LIN {X 0,Y 298.43,Z 522.305,A -85,B 0,C 180,E1 -16152.517,E2 -16152.517} C_VEL
LIN {X 0,Y 298.415,Z 522.298,A -85,B 0,C 180,E1 -16155.046,E2 -16155.046} C_VEL
LIN {X 0,Y 298.386,Z 522.319,A -85,B 0,C 180,E1 -16158.911,E2 -16158.911} C_VEL
LIN {X 0,Y 298.422,Z 522.312,A -85,B 0,C 180,E1 -16159.614,E2 -16159.614} C_VEL
LIN {X 0,Y 307.334,Z 547.466,A -85,B 0,C 180,E1 -16160.965,E2 -16160.965} C_VEL
LIN {X 0,Y 304.913,Z 622.562,A -85,B 0,C 180,E1 -16163.246,E2 -16163.246} C_VEL
LIN {X 0,Y 304.37,Z 635.953,A -85,B 0,C 180,E1 -16163.915,E2 -16163.915} C_VEL
LIN {X 0,Y 303.565,Z 648.963,A -85,B 0,C 180,E1 -16164.837,E2 -16164.837} C_VEL
LIN {X 0,Y 302.53,Z 662.384,A -85,B 0,C 180,E1 -16166.114,E2 -16166.114} C_VEL
LIN {X 0,Y 301.594,Z 672.65,A -85,B 0,C 180,E1 -16167.354,E2 -16167.354} C_VEL
LIN {X 0,Y 300.607,Z 683.859,A -85,B 0,C 180,E1 -16169.046,E2 -16169.046} C_VEL
LIN {X 0,Y 299.508,Z 693.613,A -85,B 0,C 180,E1 -16170.862,E2 -16170.862} C_VEL
LIN {X 0,Y 298.708,Z 701.527,A -85,B 0,C 180,E1 -16172.69,E2 -16172.69} C_VEL
LIN {X 0,Y 298.005,Z 709.171,A -85,B 0,C 180,E1 -16174.88,E2 -16174.88} C_VEL
LIN {X 0,Y 297.519,Z 715.25,A -85,B 0,C 180,E1 -16177.107,E2 -16177.107} C_VEL
LIN {X 0,Y 297.138,Z 719.644,A -85,B 0,C 180,E1 -16179.219,E2 -16179.219} C_VEL
LIN {X 0,Y 296.954,Z 722.708,A -85,B 0,C 180,E1 -16181.201,E2 -16181.201} C_VEL
LIN {X 0,Y 296.879,Z 725.049,A -85,B 0,C 180,E1 -16183.496,E2 -16183.496} C_VEL
LIN {X 0,Y 297.091,Z 726.196,A -85,B 0,C 180,E1 -16185.9,E2 -16185.9} C_VEL
LIN {X 0,Y 297.35,Z 726.178,A -85,B 0,C 180,E1 -16187.718,E2 -16187.718} C_VEL
LIN {X 0,Y 297.704,Z 725.653,A -85,B 0,C 180,E1 -16189.113,E2 -16189.113} C_VEL
LIN {X 0,Y 298.476,Z 723.763,A -85,B 0,C 180,E1 -16191.463,E2 -16191.463} C_VEL
LIN {X 0,Y 299.56,Z 720.269,A -85,B 0,C 180,E1 -16193.939,E2 -16193.939} C_VEL
LIN {X 0,Y 300.766,Z 716.155,A -85,B 0,C 180,E1 -16195.98,E2 -16195.98} C_VEL
LIN {X 0,Y 302.346,Z 710.28,A -85,B 0,C 180,E1 -16198.196,E2 -16198.196} C_VEL
LIN {X 0,Y 304.151,Z 702.966,A -85,B 0,C 180,E1 -16200.331,E2 -16200.331} C_VEL
LIN {X 0,Y 306.271,Z 694.292,A -85,B 0,C 180,E1 -16202.301,E2 -16202.301} C_VEL
LIN {X 0,Y 308.293,Z 684.485,A -85,B 0,C 180,E1 -16204.085,E2 -16204.085} C_VEL
LIN {X 0,Y 310.321,Z 674.239,A -85,B 0,C 180,E1 -16205.556,E2 -16205.556} C_VEL
LIN {X 0,Y 312.175,Z 663.129,A -85,B 0,C 180,E1 -16206.853,E2 -16206.853} C_VEL
LIN {X 0,Y 313.738,Z 651.807,A -85,B 0,C 180,E1 -16207.886,E2 -16207.886} C_VEL
LIN {X 0,Y 315.086,Z 638.499,A -85,B 0,C 180,E1 -16208.821,E2 -16208.821} C_VEL
LIN {X 0,Y 316.089,Z 625.669,A -85,B 0,C 180,E1 -16209.438,E2 -16209.438} C_VEL
LIN {X 0,Y 318.721,Z 584.023,A -85,B 0,C 180,E1 -16210.836,E2 -16210.836} C_VEL
LIN {X 0,Y 320.456,Z 559.213,A -85,B 0,C 180,E1 -16211.666,E2 -16211.666} C_VEL
LIN {X 0,Y 315.809,Z 550.276,A -85,B 0,C 180,E1 -16212.858,E2 -16212.858} C_VEL
LIN {X 0,Y 310.244,Z 541.034,A -85,B 0,C 180,E1 -16214.366,E2 -16214.366} C_VEL
LIN {X 0,Y 305.459,Z 533.922,A -85,B 0,C 180,E1 -16215.774,E2 -16215.774} C_VEL
LIN {X 0,Y 301.968,Z 529.251,A -85,B 0,C 180,E1 -16216.858,E2 -16216.858} C_VEL
LIN {X 0,Y 299.716,Z 526.202,A -85,B 0,C 180,E1 -16217.617,E2 -16217.617} C_VEL
LIN {X 0,Y 299.533,Z 525.763,A -85,B 0,C 180,E1 -16217.759,E2 -16217.759} C_VEL
LIN {X 0,Y 298.451,Z 522.311,A -85,B 0,C 180,E1 -16220.865,E2 -16220.865} C_VEL
LIN {X 0,Y 298.48,Z 522.303,A -85,B 0,C 180,E1 -16225.076,E2 -16225.076} C_VEL
LIN {X 0,Y 298.464,Z 522.3,A -85,B 0,C 180,E1 -16228.095,E2 -16228.095} C_VEL
LIN {X 0,Y 298.39,Z 522.313,A -85,B 0,C 180,E1 -16232.801,E2 -16232.801} C_VEL
LIN {X 0,Y 298.439,Z 522.308,A -85,B 0,C 180,E1 -16236.808,E2 -16236.808} C_VEL
LIN {X 0,Y 298.384,Z 522.319,A -85,B 0,C 180,E1 -16241.089,E2 -16241.089} C_VEL
LIN {X 0,Y 298.422,Z 522.498,A -85,B 0,C 180,E1 -16243.11,E2 -16243.11} C_VEL
LIN {X 0,Y 299.886,Z 526.896,A -85,B 0,C 180,E1 -16246.594,E2 -16246.594} C_VEL
LIN {X 0,Y 301.229,Z 531.075,A -85,B 0,C 180,E1 -16249.213,E2 -16249.213} C_VEL
LIN {X 0,Y 302.919,Z 536.463,A -85,B 0,C 180,E1 -16252.076,E2 -16252.076} C_VEL
LIN {X 0,Y 304.885,Z 544.324,A -85,B 0,C 180,E1 -16255.578,E2 -16255.578} C_VEL
LIN {X 0,Y 306.272,Z 550.468,A -85,B 0,C 180,E1 -16257.895,E2 -16257.895} C_VEL
LIN {X 0,Y 308.92,Z 555.832,A -85,B 0,C 180,E1 -16258.715,E2 -16258.715} C_VEL
LIN {X 0,Y 311.739,Z 562.313,A -85,B 0,C 180,E1 -16259.566,E2 -16259.566} C_VEL
LIN {X 0,Y 314.455,Z 576.263,A -85,B 0,C 180,E1 -16260.718,E2 -16260.718} C_VEL
LIN {X 0,Y 316.806,Z 593.122,A -85,B 0,C 180,E1 -16261.856,E2 -16261.856} C_VEL
LIN {X 0,Y 317.954,Z 609.201,A -85,B 0,C 180,E1 -16262.737,E2 -16262.737} C_VEL
LIN {X 0,Y 314.374,Z 664.551,A -85,B 0,C 180,E1 -16264.556,E2 -16264.556} C_VEL
LIN {X 0,Y 312.835,Z 678.814,A -85,B 0,C 180,E1 -16265.266,E2 -16265.266} C_VEL
LIN {X 0,Y 310.925,Z 691.732,A -85,B 0,C 180,E1 -16266.17,E2 -16266.17} C_VEL
LIN {X 0,Y 308.588,Z 705.1,A -85,B 0,C 180,E1 -16267.399,E2 -16267.399} C_VEL
LIN {X 0,Y 306.283,Z 716.906,A -85,B 0,C 180,E1 -16268.814,E2 -16268.814} C_VEL
LIN {X 0,Y 304.02,Z 727.605,A -85,B 0,C 180,E1 -16270.416,E2 -16270.416} C_VEL
LIN {X 0,Y 302.162,Z 736.378,A -85,B 0,C 180,E1 -16272.051,E2 -16272.051} C_VEL
LIN {X 0,Y 300.951,Z 742.836,A -85,B 0,C 180,E1 -16273.417,E2 -16273.417} C_VEL
LIN {X 0,Y 299.516,Z 752.316,A -85,B 0,C 180,E1 -16275.39,E2 -16275.39} C_VEL
LIN {X 0,Y 298.286,Z 759.999,A -85,B 0,C 180,E1 -16277.412,E2 -16277.412} C_VEL
LIN {X 0,Y 297.384,Z 767.055,A -85,B 0,C 180,E1 -16279.791,E2 -16279.791} C_VEL
LIN {X 0,Y 296.913,Z 771.726,A -85,B 0,C 180,E1 -16281.835,E2 -16281.835} C_VEL
LIN {X 0,Y 296.63,Z 775.891,A -85,B 0,C 180,E1 -16284.324,E2 -16284.324} C_VEL
LIN {X 0,Y 296.564,Z 777.786,A -85,B 0,C 180,E1 -16285.923,E2 -16285.923} C_VEL
LIN {X 0,Y 296.574,Z 778.942,A -85,B 0,C 180,E1 -16287.284,E2 -16287.284} C_VEL
LIN {X 0,Y 296.524,Z 779.653,A -85,B 0,C 180,E1 -16288.642,E2 -16288.642} C_VEL
LIN {X 0,Y 296.527,Z 779.976,A -85,B 0,C 180,E1 -16290,E2 -16290} C_VEL
LIN {X 0,Y 296.514,Z 779.908,A -85,B 0,C 180,E1 -16291.358,E2 -16291.358} C_VEL
LIN {X 0,Y 296.574,Z 779.416,A -85,B 0,C 180,E1 -16292.716,E2 -16292.716} C_VEL
LIN {X 0,Y 296.565,Z 778.501,A -85,B 0,C 180,E1 -16294.077,E2 -16294.077} C_VEL
LIN {X 0,Y 296.623,Z 776.953,A -85,B 0,C 180,E1 -16295.661,E2 -16295.661} C_VEL
LIN {X 0,Y 296.952,Z 773.26,A -85,B 0,C 180,E1 -16298.164,E2 -16298.164} C_VEL
LIN {X 0,Y 297.447,Z 769.078,A -85,B 0,C 180,E1 -16300.207,E2 -16300.207} C_VEL
LIN {X 0,Y 298.408,Z 762.696,A -85,B 0,C 180,E1 -16302.583,E2 -16302.583} C_VEL
LIN {X 0,Y 299.69,Z 755.711,A -85,B 0,C 180,E1 -16304.601,E2 -16304.601} C_VEL
LIN {X 0,Y 301.202,Z 747.062,A -85,B 0,C 180,E1 -16306.587,E2 -16306.587} C_VEL
LIN {X 0,Y 302.659,Z 737.985,A -85,B 0,C 180,E1 -16308.269,E2 -16308.269} C_VEL
LIN {X 0,Y 304.277,Z 728.064,A -85,B 0,C 180,E1 -16309.742,E2 -16309.742} C_VEL
LIN {X 0,Y 305.903,Z 717.021,A -85,B 0,C 180,E1 -16311.037,E2 -16311.037} C_VEL
LIN {X 0,Y 307.428,Z 704.643,A -85,B 0,C 180,E1 -16312.16,E2 -16312.16} C_VEL
LIN {X 0,Y 308.719,Z 691.932,A -85,B 0,C 180,E1 -16312.989,E2 -16312.989} C_VEL
LIN {X 0,Y 309.686,Z 678.447,A -85,B 0,C 180,E1 -16313.576,E2 -16313.576} C_VEL
LIN {X 0,Y 310.947,Z 632.674,A -85,B 0,C 180,E1 -16314.66,E2 -16314.66} C_VEL
LIN {X 0,Y 311.382,Z 606.3,A -85,B 0,C 180,E1 -16315.281,E2 -16315.281} C_VEL
LIN {X 0,Y 307.249,Z 573.521,A -85,B 0,C 180,E1 -16316.498,E2 -16316.498} C_VEL
LIN {X 0,Y 304.88,Z 559.133,A -85,B 0,C 180,E1 -16317.142,E2 -16317.142} C_VEL
LIN {X 0,Y 304.082,Z 547.632,A -85,B 0,C 180,E1 -16318.209,E2 -16318.209} C_VEL
LIN {X 0,Y 302.745,Z 542.785,A -85,B 0,C 180,E1 -16318.775,E2 -16318.775} C_VEL
LIN {X 0,Y 299.746,Z 528.657,A -85,B 0,C 180,E1 -16322.633,E2 -16322.633} C_VEL
LIN {X 0,Y 298.482,Z 522.306,A -85,B 0,C 180,E1 -16324.454,E2 -16324.454} C_VEL
LIN {X 0,Y 298.405,Z 522.277,A -85,B 0,C 180,E1 -16327.758,E2 -16327.758} C_VEL
LIN {X 0,Y 298.382,Z 522.317,A -85,B 0,C 180,E1 -16331.261,E2 -16331.261} C_VEL
LIN {X 0,Y 298.385,Z 522.314,A -85,B 0,C 180,E1 -16335.041,E2 -16335.041} C_VEL
LIN {X 0,Y 298.415,Z 522.302,A -85,B 0,C 180,E1 -16338.905,E2 -16338.905} C_VEL
LIN {X 0,Y 298.466,Z 522.292,A -85,B 0,C 180,E1 -16343.186,E2 -16343.186} C_VEL
LIN {X 0,Y 298.39,Z 522.312,A -85,B 0,C 180,E1 -16347.199,E2 -16347.199} C_VEL
LIN {X 0,Y 298.426,Z 522.3,A -85,B 0,C 180,E1 -16350.614,E2 -16350.614} C_VEL
LIN {X 0,Y 298.478,Z 522.301,A -85,B 0,C 180,E1 -16353.474,E2 -16353.474} C_VEL
LIN {X 0,Y 298.424,Z 522.288,A -85,B 0,C 180,E1 -16356.699,E2 -16356.699} C_VEL
LIN {X 0,Y 298.531,Z 522.295,A -85,B 0,C 180,E1 -16360.757,E2 -16360.757} C_VEL
LIN {X 0,Y 298.586,Z 522.274,A -85,B 0,C 180,E1 -16364.995,E2 -16364.995} C_VEL
LIN {X 0,Y 298.588,Z 522.283,A -85,B 0,C 180,E1 -16369.147,E2 -16369.147} C_VEL
LIN {X 0,Y 298.749,Z 522.242,A -85,B 0,C 180,E1 -16371.886,E2 -16371.886} C_VEL
LIN {X 0,Y 298.655,Z 522.278,A -85,B 0,C 180,E1 -16374.599,E2 -16374.599} C_VEL
LIN {X 0,Y 298.918,Z 522.229,A -85,B 0,C 180,E1 -16378.653,E2 -16378.653} C_VEL
LIN {X 0,Y 298.918,Z 522.227,A -85,B 0,C 180,E1 -16381.348,E2 -16381.348} C_VEL
LIN {X 0,Y 298.783,Z 522.25,A -85,B 0,C 180,E1 -16386.755,E2 -16386.755} C_VEL
LIN {X 0,Y 298.629,Z 522.264,A -85,B 0,C 180,E1 -16389.482,E2 -16389.482} C_VEL
LIN {X 0,Y 298.546,Z 522.292,A -85,B 0,C 180,E1 -16393.616,E2 -16393.616} C_VEL
LIN {X 0,Y 298.542,Z 522.271,A -85,B 0,C 180,E1 -16396.409,E2 -16396.409} C_VEL
LIN {X 0,Y 298.506,Z 522.302,A -85,B 0,C 180,E1 -16399.655,E2 -16399.655} C_VEL
LIN {X 0,Y 298.452,Z 522.288,A -85,B 0,C 180,E1 -16403.599,E2 -16403.599} C_VEL
LIN {X 0,Y 298.488,Z 522.304,A -85,B 0,C 180,E1 -16406.575,E2 -16406.575} C_VEL
LIN {X 0,Y 298.421,Z 522.296,A -85,B 0,C 180,E1 -16409.641,E2 -16409.641} C_VEL
LIN {X 0,Y 298.394,Z 522.318,A -85,B 0,C 180,E1 -16412.801,E2 -16412.801} C_VEL
LIN {X 0,Y 298.443,Z 522.311,A -85,B 0,C 180,E1 -16416.809,E2 -16416.809} C_VEL
LIN {X 0,Y 298.386,Z 522.32,A -85,B 0,C 180,E1 -16421.089,E2 -16421.089} C_VEL
LIN {X 0,Y 298.387,Z 522.32,A -85,B 0,C 180,E1 -16425.043,E2 -16425.043} C_VEL
LIN {X 0,Y 298.387,Z 522.315,A -85,B 0,C 180,E1 -16428.913,E2 -16428.913} C_VEL
LIN {X 0,Y 298.444,Z 522.313,A -85,B 0,C 180,E1 -16433.194,E2 -16433.194} C_VEL
LIN {X 0,Y 298.469,Z 522.372,A -85,B 0,C 180,E1 -16433.708,E2 -16433.708} C_VEL
LIN {X 0,Y 301.761,Z 534.416,A -85,B 0,C 180,E1 -16436.977,E2 -16436.977} C_VEL
LIN {X 0,Y 304.546,Z 545.909,A -85,B 0,C 180,E1 -16439.874,E2 -16439.874} C_VEL
LIN {X 0,Y 305.469,Z 550.334,A -85,B 0,C 180,E1 -16440.904,E2 -16440.904} C_VEL
LIN {X 0,Y 307.322,Z 555.912,A -85,B 0,C 180,E1 -16441.233,E2 -16441.233} C_VEL
LIN {X 0,Y 312.344,Z 582.163,A -85,B 0,C 180,E1 -16442.382,E2 -16442.382} C_VEL
LIN {X 0,Y 312.661,Z 585.629,A -85,B 0,C 180,E1 -16442.498,E2 -16442.498} C_VEL
LIN {X 0,Y 310.487,Z 661.61,A -85,B 0,C 180,E1 -16444.259,E2 -16444.259} C_VEL
LIN {X 0,Y 309.672,Z 674.686,A -85,B 0,C 180,E1 -16444.817,E2 -16444.817} C_VEL
LIN {X 0,Y 308.672,Z 686.931,A -85,B 0,C 180,E1 -16445.609,E2 -16445.609} C_VEL
LIN {X 0,Y 307.441,Z 698.55,A -85,B 0,C 180,E1 -16446.618,E2 -16446.618} C_VEL
LIN {X 0,Y 305.851,Z 709.944,A -85,B 0,C 180,E1 -16447.898,E2 -16447.898} C_VEL
LIN {X 0,Y 303.969,Z 721.329,A -85,B 0,C 180,E1 -16449.531,E2 -16449.531} C_VEL
LIN {X 0,Y 302.527,Z 729.628,A -85,B 0,C 180,E1 -16451.021,E2 -16451.021} C_VEL
LIN {X 0,Y 301.09,Z 737.273,A -85,B 0,C 180,E1 -16452.687,E2 -16452.687} C_VEL
LIN {X 0,Y 299.86,Z 744.718,A -85,B 0,C 180,E1 -16454.712,E2 -16454.712} C_VEL
LIN {X 0,Y 298.518,Z 751.584,A -85,B 0,C 180,E1 -16457.076,E2 -16457.076} C_VEL
LIN {X 0,Y 297.694,Z 756.111,A -85,B 0,C 180,E1 -16459.114,E2 -16459.114} C_VEL
LIN {X 0,Y 297.33,Z 758.491,A -85,B 0,C 180,E1 -16460.476,E2 -16460.476} C_VEL
LIN {X 0,Y 297.01,Z 760.426,A -85,B 0,C 180,E1 -16461.838,E2 -16461.838} C_VEL
LIN {X 0,Y 296.669,Z 762.838,A -85,B 0,C 180,E1 -16464.256,E2 -16464.256} C_VEL
LIN {X 0,Y 296.596,Z 763.726,A -85,B 0,C 180,E1 -16465.924,E2 -16465.924} C_VEL
LIN {X 0,Y 296.563,Z 764.025,A -85,B 0,C 180,E1 -16467.283,E2 -16467.283} C_VEL
LIN {X 0,Y 296.509,Z 763.946,A -85,B 0,C 180,E1 -16468.642,E2 -16468.642} C_VEL
LIN {X 0,Y 296.524,Z 763.439,A -85,B 0,C 180,E1 -16470,E2 -16470} C_VEL
LIN {X 0,Y 296.753,Z 761.245,A -85,B 0,C 180,E1 -16472.715,E2 -16472.715} C_VEL
LIN {X 0,Y 297.138,Z 758.502,A -85,B 0,C 180,E1 -16474.748,E2 -16474.748} C_VEL
LIN {X 0,Y 297.61,Z 754.749,A -85,B 0,C 180,E1 -16476.781,E2 -16476.781} C_VEL
LIN {X 0,Y 298.284,Z 749.88,A -85,B 0,C 180,E1 -16478.809,E2 -16478.809} C_VEL
LIN {X 0,Y 299.248,Z 743.742,A -85,B 0,C 180,E1 -16480.829,E2 -16480.829} C_VEL
LIN {X 0,Y 300.514,Z 736.035,A -85,B 0,C 180,E1 -16482.836,E2 -16482.836} C_VEL
LIN {X 0,Y 302.039,Z 726.445,A -85,B 0,C 180,E1 -16484.83,E2 -16484.83} C_VEL
LIN {X 0,Y 303.5,Z 716.427,A -85,B 0,C 180,E1 -16486.479,E2 -16486.479} C_VEL
LIN {X 0,Y 304.859,Z 706.554,A -85,B 0,C 180,E1 -16487.785,E2 -16487.785} C_VEL
LIN {X 0,Y 306.131,Z 695.827,A -85,B 0,C 180,E1 -16488.921,E2 -16488.921} C_VEL
LIN {X 0,Y 307.336,Z 684.004,A -85,B 0,C 180,E1 -16489.886,E2 -16489.886} C_VEL
LIN {X 0,Y 308.202,Z 670.49,A -85,B 0,C 180,E1 -16490.679,E2 -16490.679} C_VEL
LIN {X 0,Y 308.801,Z 657.426,A -85,B 0,C 180,E1 -16491.165,E2 -16491.165} C_VEL
LIN {X 0,Y 310.66,Z 582.64,A -85,B 0,C 180,E1 -16492.878,E2 -16492.878} C_VEL
LIN {X 0,Y 305.83,Z 555.571,A -85,B 0,C 180,E1 -16493.97,E2 -16493.97} C_VEL
LIN {X 0,Y 304.741,Z 550.103,A -85,B 0,C 180,E1 -16494.227,E2 -16494.227} C_VEL
LIN {X 0,Y 302.942,Z 540.186,A -85,B 0,C 180,E1 -16496.523,E2 -16496.523} C_VEL
LIN {X 0,Y 300.186,Z 528.619,A -85,B 0,C 180,E1 -16499.449,E2 -16499.449} C_VEL
LIN {X 0,Y 298.436,Z 522.311,A -85,B 0,C 180,E1 -16501.105,E2 -16501.105} C_VEL
LIN {X 0,Y 298.429,Z 522.31,A -85,B 0,C 180,E1 -16504.486,E2 -16504.486} C_VEL
LIN {X 0,Y 298.439,Z 522.31,A -85,B 0,C 180,E1 -16507.753,E2 -16507.753} C_VEL
LIN {X 0,Y 298.451,Z 522.302,A -85,B 0,C 180,E1 -16511.249,E2 -16511.249} C_VEL
LIN {X 0,Y 298.43,Z 522.305,A -85,B 0,C 180,E1 -16512.517,E2 -16512.517} C_VEL
LIN {X 0,Y 297.789,Z 522.392,A -85,B 0,C 180,E1 -16513.644,E2 -16513.644} C_VEL
LIN {X 0,Y 294.902,Z 522.755,A -85,B 0,C 180,E1 -16515.477,E2 -16515.477} C_VEL
LIN {X 0,Y 292.443,Z 523.06,A -85,B 0,C 180,E1 -16516.965,E2 -16516.965} C_VEL
LIN {X 0,Y 291.406,Z 523.188,A -85,B 0,C 180,E1 -16518.12,E2 -16518.12} C_VEL
LIN {X 0,Y 291.332,Z 523.197,A -85,B 0,C 180,E1 -16518.511,E2 -16518.511} C_VEL
LIN {X 0,Y 291.376,Z 523.213,A -85,B 0,C 180,E1 -16519.245,E2 -16519.245} C_VEL
LIN {X 0,Y 300.482,Z 548.952,A -85,B 0,C 180,E1 -16520.636,E2 -16520.636} C_VEL
LIN {X 0,Y 297.989,Z 623.073,A -85,B 0,C 180,E1 -16522.971,E2 -16522.971} C_VEL
LIN {X 0,Y 297.42,Z 636.511,A -85,B 0,C 180,E1 -16523.662,E2 -16523.662} C_VEL
LIN {X 0,Y 296.587,Z 649.592,A -85,B 0,C 180,E1 -16524.614,E2 -16524.614} C_VEL
LIN {X 0,Y 295.526,Z 662.981,A -85,B 0,C 180,E1 -16525.918,E2 -16525.918} C_VEL
LIN {X 0,Y 294.459,Z 674.144,A -85,B 0,C 180,E1 -16527.316,E2 -16527.316} C_VEL
LIN {X 0,Y 293.481,Z 685.006,A -85,B 0,C 180,E1 -16529.012,E2 -16529.012} C_VEL
LIN {X 0,Y 292.394,Z 694.638,A -85,B 0,C 180,E1 -16530.874,E2 -16530.874} C_VEL
LIN {X 0,Y 291.587,Z 702.483,A -85,B 0,C 180,E1 -16532.745,E2 -16532.745} C_VEL
LIN {X 0,Y 290.91,Z 710.082,A -85,B 0,C 180,E1 -16534.989,E2 -16534.989} C_VEL
LIN {X 0,Y 290.409,Z 715.961,A -85,B 0,C 180,E1 -16537.219,E2 -16537.219} C_VEL
LIN {X 0,Y 290.016,Z 720.414,A -85,B 0,C 180,E1 -16539.428,E2 -16539.428} C_VEL
LIN {X 0,Y 289.84,Z 723.632,A -85,B 0,C 180,E1 -16541.625,E2 -16541.625} C_VEL
LIN {X 0,Y 289.785,Z 725.16,A -85,B 0,C 180,E1 -16543.08,E2 -16543.08} C_VEL
LIN {X 0,Y 289.855,Z 726.195,A -85,B 0,C 180,E1 -16544.531,E2 -16544.531} C_VEL
LIN {X 0,Y 290.049,Z 726.754,A -85,B 0,C 180,E1 -16545.977,E2 -16545.977} C_VEL
LIN {X 0,Y 290.242,Z 726.895,A -85,B 0,C 180,E1 -16547.412,E2 -16547.412} C_VEL
LIN {X 0,Y 290.554,Z 726.57,A -85,B 0,C 180,E1 -16548.842,E2 -16548.842} C_VEL
LIN {X 0,Y 291.417,Z 724.833,A -85,B 0,C 180,E1 -16551.401,E2 -16551.401} C_VEL
LIN {X 0,Y 292.445,Z 721.882,A -85,B 0,C 180,E1 -16553.791,E2 -16553.791} C_VEL
LIN {X 0,Y 293.682,Z 718.135,A -85,B 0,C 180,E1 -16555.883,E2 -16555.883} C_VEL
LIN {X 0,Y 295.321,Z 712.655,A -85,B 0,C 180,E1 -16558.16,E2 -16558.16} C_VEL
LIN {X 0,Y 297.181,Z 705.802,A -85,B 0,C 180,E1 -16560.338,E2 -16560.338} C_VEL
LIN {X 0,Y 299.304,Z 697.709,A -85,B 0,C 180,E1 -16562.355,E2 -16562.355} C_VEL
LIN {X 0,Y 301.648,Z 687.639,A -85,B 0,C 180,E1 -16564.342,E2 -16564.342} C_VEL
LIN {X 0,Y 303.8,Z 677.756,A -85,B 0,C 180,E1 -16565.889,E2 -16565.889} C_VEL
LIN {X 0,Y 305.772,Z 666.848,A -85,B 0,C 180,E1 -16567.256,E2 -16567.256} C_VEL
LIN {X 0,Y 307.574,Z 655.47,A -85,B 0,C 180,E1 -16568.376,E2 -16568.376} C_VEL
LIN {X 0,Y 309.044,Z 643.218,A -85,B 0,C 180,E1 -16569.325,E2 -16569.325} C_VEL
LIN {X 0,Y 310.182,Z 630.027,A -85,B 0,C 180,E1 -16570.072,E2 -16570.072} C_VEL
LIN {X 0,Y 311.917,Z 603.449,A -85,B 0,C 180,E1 -16571.032,E2 -16571.032} C_VEL
LIN {X 0,Y 315.065,Z 561.977,A -85,B 0,C 180,E1 -16572.426,E2 -16572.426} C_VEL
LIN {X 0,Y 310.055,Z 552.454,A -85,B 0,C 180,E1 -16573.818,E2 -16573.818} C_VEL
LIN {X 0,Y 304.716,Z 543.622,A -85,B 0,C 180,E1 -16575.389,E2 -16575.389} C_VEL
LIN {X 0,Y 301.575,Z 539.128,A -85,B 0,C 180,E1 -16576.351,E2 -16576.351} C_VEL
LIN {X 0,Y 298.77,Z 535.196,A -85,B 0,C 180,E1 -16577.297,E2 -16577.297} C_VEL
LIN {X 0,Y 295.688,Z 531.254,A -85,B 0,C 180,E1 -16578.358,E2 -16578.358} C_VEL
LIN {X 0,Y 293.052,Z 527.899,A -85,B 0,C 180,E1 -16579.367,E2 -16579.367} C_VEL
LIN {X 0,Y 292.655,Z 527.207,A -85,B 0,C 180,E1 -16579.554,E2 -16579.554} C_VEL
LIN {X 0,Y 291.629,Z 524.342,A -85,B 0,C 180,E1 -16582.68,E2 -16582.68} C_VEL
LIN {X 0,Y 291.394,Z 523.185,A -85,B 0,C 180,E1 -16584.206,E2 -16584.206} C_VEL
LIN {X 0,Y 291.42,Z 523.179,A -85,B 0,C 180,E1 -16587.272,E2 -16587.272} C_VEL
LIN {X 0,Y 291.332,Z 523.189,A -85,B 0,C 180,E1 -16590.437,E2 -16590.437} C_VEL
LIN {X 0,Y 291.339,Z 523.188,A -85,B 0,C 180,E1 -16593.699,E2 -16593.699} C_VEL
LIN {X 0,Y 291.368,Z 523.192,A -85,B 0,C 180,E1 -16597.254,E2 -16597.254} C_VEL
LIN {X 0,Y 291.355,Z 523.201,A -85,B 0,C 180,E1 -16599.679,E2 -16599.679} C_VEL
LIN {X 0,Y 292.076,Z 525.522,A -85,B 0,C 180,E1 -16602.356,E2 -16602.356} C_VEL
LIN {X 0,Y 293.554,Z 529.815,A -85,B 0,C 180,E1 -16606.031,E2 -16606.031} C_VEL
LIN {X 0,Y 295.296,Z 535.352,A -85,B 0,C 180,E1 -16609.605,E2 -16609.605} C_VEL
LIN {X 0,Y 297.112,Z 541.628,A -85,B 0,C 180,E1 -16612.903,E2 -16612.903} C_VEL
LIN {X 0,Y 298.857,Z 548.989,A -85,B 0,C 180,E1 -16616.141,E2 -16616.141} C_VEL
LIN {X 0,Y 301.594,Z 554.384,A -85,B 0,C 180,E1 -16617.094,E2 -16617.094} C_VEL
LIN {X 0,Y 305.364,Z 562.266,A -85,B 0,C 180,E1 -16618.337,E2 -16618.337} C_VEL
LIN {X 0,Y 307.021,Z 566.083,A -85,B 0,C 180,E1 -16618.866,E2 -16618.866} C_VEL
LIN {X 0,Y 309.812,Z 581.74,A -85,B 0,C 180,E1 -16620.17,E2 -16620.17} C_VEL
LIN {X 0,Y 311.638,Z 597.066,A -85,B 0,C 180,E1 -16621.212,E2 -16621.212} C_VEL
LIN {X 0,Y 312.462,Z 610.29,A -85,B 0,C 180,E1 -16621.942,E2 -16621.942} C_VEL
LIN {X 0,Y 308.562,Z 665.089,A -85,B 0,C 180,E1 -16623.814,E2 -16623.814} C_VEL
LIN {X 0,Y 307.037,Z 678.326,A -85,B 0,C 180,E1 -16624.494,E2 -16624.494} C_VEL
LIN {X 0,Y 304.875,Z 692.132,A -85,B 0,C 180,E1 -16625.485,E2 -16625.485} C_VEL
LIN {X 0,Y 302.72,Z 703.718,A -85,B 0,C 180,E1 -16626.574,E2 -16626.574} C_VEL
LIN {X 0,Y 300.52,Z 714.387,A -85,B 0,C 180,E1 -16627.846,E2 -16627.846} C_VEL
LIN {X 0,Y 297.84,Z 726.332,A -85,B 0,C 180,E1 -16629.632,E2 -16629.632} C_VEL
LIN {X 0,Y 295.766,Z 735.251,A -85,B 0,C 180,E1 -16631.29,E2 -16631.29} C_VEL
LIN {X 0,Y 293.634,Z 745.835,A -85,B 0,C 180,E1 -16633.667,E2 -16633.667} C_VEL
LIN {X 0,Y 292.404,Z 753.434,A -85,B 0,C 180,E1 -16635.383,E2 -16635.383} C_VEL
LIN {X 0,Y 291.139,Z 760.858,A -85,B 0,C 180,E1 -16637.452,E2 -16637.452} C_VEL
LIN {X 0,Y 290.383,Z 766.811,A -85,B 0,C 180,E1 -16639.542,E2 -16639.542} C_VEL
LIN {X 0,Y 289.863,Z 771.493,A -85,B 0,C 180,E1 -16641.635,E2 -16641.635} C_VEL
LIN {X 0,Y 289.578,Z 775.046,A -85,B 0,C 180,E1 -16643.73,E2 -16643.73} C_VEL
LIN {X 0,Y 289.466,Z 777.573,A -85,B 0,C 180,E1 -16645.823,E2 -16645.823} C_VEL
LIN {X 0,Y 289.499,Z 778.739,A -85,B 0,C 180,E1 -16647.217,E2 -16647.217} C_VEL
LIN {X 0,Y 289.444,Z 779.456,A -85,B 0,C 180,E1 -16648.609,E2 -16648.609} C_VEL
LIN {X 0,Y 289.444,Z 779.783,A -85,B 0,C 180,E1 -16650,E2 -16650} C_VEL
LIN {X 0,Y 289.435,Z 779.72,A -85,B 0,C 180,E1 -16651.391,E2 -16651.391} C_VEL
LIN {X 0,Y 289.499,Z 779.238,A -85,B 0,C 180,E1 -16652.783,E2 -16652.783} C_VEL
LIN {X 0,Y 289.516,Z 777.021,A -85,B 0,C 180,E1 -16655.572,E2 -16655.572} C_VEL
LIN {X 0,Y 289.742,Z 774.251,A -85,B 0,C 180,E1 -16657.666,E2 -16657.666} C_VEL
LIN {X 0,Y 290.241,Z 770.451,A -85,B 0,C 180,E1 -16659.759,E2 -16659.759} C_VEL
LIN {X 0,Y 290.957,Z 765.509,A -85,B 0,C 180,E1 -16661.848,E2 -16661.848} C_VEL
LIN {X 0,Y 292.089,Z 759.284,A -85,B 0,C 180,E1 -16663.922,E2 -16663.922} C_VEL
LIN {X 0,Y 293.505,Z 751.477,A -85,B 0,C 180,E1 -16665.984,E2 -16665.984} C_VEL
LIN {X 0,Y 295.026,Z 743.072,A -85,B 0,C 180,E1 -16667.769,E2 -16667.769} C_VEL
LIN {X 0,Y 296.593,Z 733.767,A -85,B 0,C 180,E1 -16669.374,E2 -16669.374} C_VEL
LIN {X 0,Y 298.454,Z 722.857,A -85,B 0,C 180,E1 -16670.864,E2 -16670.864} C_VEL
LIN {X 0,Y 299.975,Z 712.158,A -85,B 0,C 180,E1 -16672.015,E2 -16672.015} C_VEL
LIN {X 0,Y 301.401,Z 700.379,A -85,B 0,C 180,E1 -16672.99,E2 -16672.99} C_VEL
LIN {X 0,Y 302.592,Z 687.594,A -85,B 0,C 180,E1 -16673.754,E2 -16673.754} C_VEL
LIN {X 0,Y 303.437,Z 675.041,A -85,B 0,C 180,E1 -16674.229,E2 -16674.229} C_VEL
LIN {X 0,Y 305.091,Z 607.869,A -85,B 0,C 180,E1 -16675.821,E2 -16675.821} C_VEL
LIN {X 0,Y 300.957,Z 574.656,A -85,B 0,C 180,E1 -16677.089,E2 -16677.089} C_VEL
LIN {X 0,Y 298.435,Z 559.219,A -85,B 0,C 180,E1 -16677.782,E2 -16677.782} C_VEL
LIN {X 0,Y 297.976,Z 551.255,A -85,B 0,C 180,E1 -16678.553,E2 -16678.553} C_VEL
LIN {X 0,Y 296.084,Z 544.299,A -85,B 0,C 180,E1 -16679.387,E2 -16679.387} C_VEL
LIN {X 0,Y 294.896,Z 540.06,A -85,B 0,C 180,E1 -16679.936,E2 -16679.936} C_VEL
LIN {X 0,Y 291.912,Z 525.529,A -85,B 0,C 180,E1 -16684.031,E2 -16684.031} C_VEL
LIN {X 0,Y 291.411,Z 523.187,A -85,B 0,C 180,E1 -16684.723,E2 -16684.723} C_VEL
LIN {X 0,Y 291.369,Z 523.156,A -85,B 0,C 180,E1 -16687.252,E2 -16687.252} C_VEL
LIN {X 0,Y 291.33,Z 523.19,A -85,B 0,C 180,E1 -16690.642,E2 -16690.642} C_VEL
LIN {X 0,Y 291.31,Z 523.191,A -85,B 0,C 180,E1 -16694.397,E2 -16694.397} C_VEL
LIN {X 0,Y 291.352,Z 523.18,A -85,B 0,C 180,E1 -16698.397,E2 -16698.397} C_VEL
LIN {X 0,Y 291.376,Z 523.191,A -85,B 0,C 180,E1 -16701.162,E2 -16701.162} C_VEL
LIN {X 0,Y 291.381,Z 523.18,A -85,B 0,C 180,E1 -16704.629,E2 -16704.629} C_VEL
LIN {X 0,Y 291.367,Z 523.182,A -85,B 0,C 180,E1 -16707.95,E2 -16707.95} C_VEL
LIN {X 0,Y 291.377,Z 523.182,A -85,B 0,C 180,E1 -16711.158,E2 -16711.158} C_VEL
LIN {X 0,Y 291.41,Z 523.176,A -85,B 0,C 180,E1 -16714.272,E2 -16714.272} C_VEL
LIN {X 0,Y 291.368,Z 523.172,A -85,B 0,C 180,E1 -16717.299,E2 -16717.299} C_VEL
LIN {X 0,Y 291.452,Z 523.178,A -85,B 0,C 180,E1 -16720.27,E2 -16720.27} C_VEL
LIN {X 0,Y 291.534,Z 523.149,A -85,B 0,C 180,E1 -16724.634,E2 -16724.634} C_VEL
LIN {X 0,Y 291.532,Z 523.165,A -85,B 0,C 180,E1 -16728.881,E2 -16728.881} C_VEL
LIN {X 0,Y 291.7,Z 523.119,A -85,B 0,C 180,E1 -16731.688,E2 -16731.688} C_VEL
LIN {X 0,Y 291.625,Z 523.153,A -85,B 0,C 180,E1 -16734.469,E2 -16734.469} C_VEL
LIN {X 0,Y 291.884,Z 523.105,A -85,B 0,C 180,E1 -16738.621,E2 -16738.621} C_VEL
LIN {X 0,Y 291.885,Z 523.103,A -85,B 0,C 180,E1 -16741.38,E2 -16741.38} C_VEL
LIN {X 0,Y 291.731,Z 523.126,A -85,B 0,C 180,E1 -16746.919,E2 -16746.919} C_VEL
LIN {X 0,Y 291.569,Z 523.146,A -85,B 0,C 180,E1 -16749.714,E2 -16749.714} C_VEL
LIN {X 0,Y 291.516,Z 523.166,A -85,B 0,C 180,E1 -16753.951,E2 -16753.951} C_VEL
LIN {X 0,Y 291.481,Z 523.151,A -85,B 0,C 180,E1 -16756.819,E2 -16756.819} C_VEL
LIN {X 0,Y 291.446,Z 523.18,A -85,B 0,C 180,E1 -16759.876,E2 -16759.876} C_VEL
LIN {X 0,Y 291.395,Z 523.171,A -85,B 0,C 180,E1 -16764.206,E2 -16764.206} C_VEL
LIN {X 0,Y 291.424,Z 523.182,A -85,B 0,C 180,E1 -16767.272,E2 -16767.272} C_VEL
LIN {X 0,Y 291.337,Z 523.182,A -85,B 0,C 180,E1 -16770.437,E2 -16770.437} C_VEL
LIN {X 0,Y 291.342,Z 523.188,A -85,B 0,C 180,E1 -16773.699,E2 -16773.699} C_VEL
LIN {X 0,Y 291.374,Z 523.196,A -85,B 0,C 180,E1 -16777.255,E2 -16777.255} C_VEL
LIN {X 0,Y 291.331,Z 523.194,A -85,B 0,C 180,E1 -16780.643,E2 -16780.643} C_VEL
LIN {X 0,Y 291.312,Z 523.197,A -85,B 0,C 180,E1 -16784.398,E2 -16784.398} C_VEL
LIN {X 0,Y 291.326,Z 523.198,A -85,B 0,C 180,E1 -16788.405,E2 -16788.405} C_VEL
LIN {X 0,Y 291.347,Z 523.194,A -85,B 0,C 180,E1 -16791.159,E2 -16791.159} C_VEL
LIN {X 0,Y 291.398,Z 523.202,A -85,B 0,C 180,E1 -16792.989,E2 -16792.989} C_VEL
LIN {X 0,Y 294.94,Z 535.888,A -85,B 0,C 180,E1 -16796.513,E2 -16796.513} C_VEL
LIN {X 0,Y 298.221,Z 549.592,A -85,B 0,C 180,E1 -16799.993,E2 -16799.993} C_VEL
LIN {X 0,Y 298.422,Z 550.512,A -85,B 0,C 180,E1 -16800.184,E2 -16800.184} C_VEL
LIN {X 0,Y 301.098,Z 557.468,A -85,B 0,C 180,E1 -16800.649,E2 -16800.649} C_VEL
LIN {X 0,Y 306.145,Z 583.989,A -85,B 0,C 180,E1 -16801.846,E2 -16801.846} C_VEL
LIN {X 0,Y 306.194,Z 590.92,A -85,B 0,C 180,E1 -16802.03,E2 -16802.03} C_VEL
LIN {X 0,Y 304.103,Z 660.912,A -85,B 0,C 180,E1 -16803.677,E2 -16803.677} C_VEL
LIN {X 0,Y 303.312,Z 673.642,A -85,B 0,C 180,E1 -16804.204,E2 -16804.204} C_VEL
LIN {X 0,Y 302.348,Z 685.268,A -85,B 0,C 180,E1 -16804.937,E2 -16804.937} C_VEL
LIN {X 0,Y 301.074,Z 697.261,A -85,B 0,C 180,E1 -16805.964,E2 -16805.964} C_VEL
LIN {X 0,Y 299.477,Z 708.638,A -85,B 0,C 180,E1 -16807.219,E2 -16807.219} C_VEL
LIN {X 0,Y 297.922,Z 718.225,A -85,B 0,C 180,E1 -16808.553,E2 -16808.553} C_VEL
LIN {X 0,Y 296.111,Z 727.94,A -85,B 0,C 180,E1 -16810.232,E2 -16810.232} C_VEL
LIN {X 0,Y 294.273,Z 737.353,A -85,B 0,C 180,E1 -16812.273,E2 -16812.273} C_VEL
LIN {X 0,Y 292.949,Z 744.823,A -85,B 0,C 180,E1 -16814.342,E2 -16814.342} C_VEL
LIN {X 0,Y 291.99,Z 749.93,A -85,B 0,C 180,E1 -16816.073,E2 -16816.073} C_VEL
LIN {X 0,Y 290.939,Z 754.854,A -85,B 0,C 180,E1 -16818.152,E2 -16818.152} C_VEL
LIN {X 0,Y 290.298,Z 758.642,A -85,B 0,C 180,E1 -16820.243,E2 -16820.243} C_VEL
LIN {X 0,Y 289.967,Z 760.583,A -85,B 0,C 180,E1 -16821.638,E2 -16821.638} C_VEL
LIN {X 0,Y 289.597,Z 763.127,A -85,B 0,C 180,E1 -16824.273,E2 -16824.273} C_VEL
LIN {X 0,Y 289.497,Z 763.909,A -85,B 0,C 180,E1 -16825.824,E2 -16825.824} C_VEL
LIN {X 0,Y 289.491,Z 764.213,A -85,B 0,C 180,E1 -16827.217,E2 -16827.217} C_VEL
LIN {X 0,Y 289.43,Z 764.14,A -85,B 0,C 180,E1 -16828.609,E2 -16828.609} C_VEL
LIN {X 0,Y 289.441,Z 763.645,A -85,B 0,C 180,E1 -16830,E2 -16830} C_VEL
LIN {X 0,Y 289.681,Z 761.463,A -85,B 0,C 180,E1 -16832.781,E2 -16832.781} C_VEL
LIN {X 0,Y 290.088,Z 758.732,A -85,B 0,C 180,E1 -16834.864,E2 -16834.864} C_VEL
LIN {X 0,Y 290.553,Z 754.993,A -85,B 0,C 180,E1 -16836.946,E2 -16836.946} C_VEL
LIN {X 0,Y 291.274,Z 750.137,A -85,B 0,C 180,E1 -16839.023,E2 -16839.023} C_VEL
LIN {X 0,Y 292.279,Z 744.018,A -85,B 0,C 180,E1 -16841.09,E2 -16841.09} C_VEL
LIN {X 0,Y 293.626,Z 736.332,A -85,B 0,C 180,E1 -16843.143,E2 -16843.143} C_VEL
LIN {X 0,Y 295.207,Z 726.762,A -85,B 0,C 180,E1 -16845.181,E2 -16845.181} C_VEL
LIN {X 0,Y 296.73,Z 716.781,A -85,B 0,C 180,E1 -16846.866,E2 -16846.866} C_VEL
LIN {X 0,Y 298.327,Z 705.568,A -85,B 0,C 180,E1 -16848.366,E2 -16848.366} C_VEL
LIN {X 0,Y 299.615,Z 694.555,A -85,B 0,C 180,E1 -16849.527,E2 -16849.527} C_VEL
LIN {X 0,Y 300.812,Z 683.325,A -85,B 0,C 180,E1 -16850.425,E2 -16850.425} C_VEL
LIN {X 0,Y 301.641,Z 670.512,A -85,B 0,C 180,E1 -16851.184,E2 -16851.184} C_VEL
LIN {X 0,Y 302.266,Z 657.266,A -85,B 0,C 180,E1 -16851.68,E2 -16851.68} C_VEL
LIN {X 0,Y 304.162,Z 583.685,A -85,B 0,C 180,E1 -16853.399,E2 -16853.399} C_VEL
LIN {X 0,Y 299.561,Z 557.431,A -85,B 0,C 180,E1 -16854.485,E2 -16854.485} C_VEL
LIN {X 0,Y 297.973,Z 550.905,A -85,B 0,C 180,E1 -16854.804,E2 -16854.804} C_VEL
LIN {X 0,Y 297.748,Z 550.008,A -85,B 0,C 180,E1 -16854.906,E2 -16854.906} C_VEL
LIN {X 0,Y 295.307,Z 538.033,A -85,B 0,C 180,E1 -16857.786,E2 -16857.786} C_VEL
LIN {X 0,Y 292.412,Z 526.93,A -85,B 0,C 180,E1 -16860.712,E2 -16860.712} C_VEL
LIN {X 0,Y 291.362,Z 523.193,A -85,B 0,C 180,E1 -16861.744,E2 -16861.744} C_VEL
LIN {X 0,Y 291.386,Z 523.189,A -85,B 0,C 180,E1 -16865.37,E2 -16865.37} C_VEL
LIN {X 0,Y 291.378,Z 523.189,A -85,B 0,C 180,E1 -16868.837,E2 -16868.837} C_VEL
LIN {X 0,Y 291.396,Z 523.189,A -85,B 0,C 180,E1 -16872.497,E2 -16872.497} C_VEL
LIN {X 0,Y 291.345,Z 523.184,A -85,B 0,C 180,E1 -16876.357,E2 -16876.357} C_VEL
LIN {X 0,Y 291.332,Z 523.197,A -85,B 0,C 180,E1 -16878.511,E2 -16878.511} C_VEL
LIN {X 0,Y 291.862,Z 523.938,A -85,B 0,C 180,E1 -16878.985,E2 -16878.985} C_VEL
LIN {X 0,Y 293.387,Z 526.274,A -85,B 0,C 180,E1 -16879.44,E2 -16879.44} C_VEL
LIN {X 0,Y 295.583,Z 530.447,A -85,B 0,C 180,E1 -16879.742,E2 -16879.742} C_VEL
LIN {X 0,Y 296.524,Z 534.294,A -85,B 0,C 180,E1 -16879.926,E2 -16879.926} C_VEL
LIN {X 0,Y 296.313,Z 539.044,A -85,B 0,C 180,E1 -16880.045,E2 -16880.045} C_VEL
LIN {X 0,Y 293.571,Z 551.983,A -85,B 0,C 180,E1 -16880.365,E2 -16880.365} C_VEL
LIN {X 0,Y 293.5,Z 553.177,A -85,B 0,C 180,E1 -16880.403,E2 -16880.403} C_VEL
LIN {X 0,Y 291.062,Z 623.382,A -85,B 0,C 180,E1 -16882.677,E2 -16882.677} C_VEL
LIN {X 0,Y 290.431,Z 637.502,A -85,B 0,C 180,E1 -16883.423,E2 -16883.423} C_VEL
LIN {X 0,Y 289.587,Z 650.192,A -85,B 0,C 180,E1 -16884.376,E2 -16884.376} C_VEL
LIN {X 0,Y 288.658,Z 661.851,A -85,B 0,C 180,E1 -16885.523,E2 -16885.523} C_VEL
LIN {X 0,Y 287.668,Z 672.733,A -85,B 0,C 180,E1 -16886.862,E2 -16886.862} C_VEL
LIN {X 0,Y 286.704,Z 682.84,A -85,B 0,C 180,E1 -16888.401,E2 -16888.401} C_VEL
LIN {X 0,Y 285.66,Z 692.156,A -85,B 0,C 180,E1 -16890.135,E2 -16890.135} C_VEL
LIN {X 0,Y 284.786,Z 700.532,A -85,B 0,C 180,E1 -16892.037,E2 -16892.037} C_VEL
LIN {X 0,Y 284.107,Z 707.433,A -85,B 0,C 180,E1 -16893.954,E2 -16893.954} C_VEL
LIN {X 0,Y 283.611,Z 713.053,A -85,B 0,C 180,E1 -16895.866,E2 -16895.866} C_VEL
LIN {X 0,Y 283.119,Z 718.385,A -85,B 0,C 180,E1 -16898.139,E2 -16898.139} C_VEL
LIN {X 0,Y 282.807,Z 722.901,A -85,B 0,C 180,E1 -16900.788,E2 -16900.788} C_VEL
LIN {X 0,Y 282.698,Z 725.139,A -85,B 0,C 180,E1 -16902.643,E2 -16902.643} C_VEL
LIN {X 0,Y 282.74,Z 726.385,A -85,B 0,C 180,E1 -16904.131,E2 -16904.131} C_VEL
LIN {X 0,Y 282.92,Z 727.204,A -85,B 0,C 180,E1 -16905.644,E2 -16905.644} C_VEL
LIN {X 0,Y 283.114,Z 727.502,A -85,B 0,C 180,E1 -16907.09,E2 -16907.09} C_VEL
LIN {X 0,Y 283.427,Z 727.37,A -85,B 0,C 180,E1 -16908.558,E2 -16908.558} C_VEL
LIN {X 0,Y 283.865,Z 726.814,A -85,B 0,C 180,E1 -16910.019,E2 -16910.019} C_VEL
LIN {X 0,Y 284.386,Z 725.794,A -85,B 0,C 180,E1 -16911.473,E2 -16911.473} C_VEL
LIN {X 0,Y 284.973,Z 724.333,A -85,B 0,C 180,E1 -16912.916,E2 -16912.916} C_VEL
LIN {X 0,Y 286.153,Z 721.272,A -85,B 0,C 180,E1 -16915.068,E2 -16915.068} C_VEL
LIN {X 0,Y 287.563,Z 717.109,A -85,B 0,C 180,E1 -16917.198,E2 -16917.198} C_VEL
LIN {X 0,Y 289.215,Z 711.742,A -85,B 0,C 180,E1 -16919.304,E2 -16919.304} C_VEL
LIN {X 0,Y 291.199,Z 705.041,A -85,B 0,C 180,E1 -16921.383,E2 -16921.383} C_VEL
LIN {X 0,Y 293.55,Z 696.588,A -85,B 0,C 180,E1 -16923.431,E2 -16923.431} C_VEL
LIN {X 0,Y 295.649,Z 688.006,A -85,B 0,C 180,E1 -16925.114,E2 -16925.114} C_VEL
LIN {X 0,Y 297.827,Z 678.567,A -85,B 0,C 180,E1 -16926.605,E2 -16926.605} C_VEL
LIN {X 0,Y 299.8,Z 668.467,A -85,B 0,C 180,E1 -16927.918,E2 -16927.918} C_VEL
LIN {X 0,Y 301.955,Z 655.776,A -85,B 0,C 180,E1 -16929.208,E2 -16929.208} C_VEL
LIN {X 0,Y 303.518,Z 643.458,A -85,B 0,C 180,E1 -16930.169,E2 -16930.169} C_VEL
LIN {X 0,Y 304.732,Z 630.126,A -85,B 0,C 180,E1 -16930.926,E2 -16930.926} C_VEL
LIN {X 0,Y 306.971,Z 598.971,A -85,B 0,C 180,E1 -16932.058,E2 -16932.058} C_VEL
LIN {X 0,Y 309.694,Z 564.512,A -85,B 0,C 180,E1 -16933.275,E2 -16933.275} C_VEL
LIN {X 0,Y 304.551,Z 554.913,A -85,B 0,C 180,E1 -16934.794,E2 -16934.794} C_VEL
LIN {X 0,Y 298.902,Z 545.725,A -85,B 0,C 180,E1 -16936.602,E2 -16936.602} C_VEL
LIN {X 0,Y 295.087,Z 540.517,A -85,B 0,C 180,E1 -16937.912,E2 -16937.912} C_VEL
LIN {X 0,Y 292.47,Z 537.054,A -85,B 0,C 180,E1 -16938.892,E2 -16938.892} C_VEL
LIN {X 0,Y 289.223,Z 532.959,A -85,B 0,C 180,E1 -16940.187,E2 -16940.187} C_VEL
LIN {X 0,Y 286.107,Z 529.192,A -85,B 0,C 180,E1 -16941.582,E2 -16941.582} C_VEL
LIN {X 0,Y 285.8,Z 528.644,A -85,B 0,C 180,E1 -16941.835,E2 -16941.835} C_VEL
LIN {X 0,Y 285.135,Z 526.511,A -85,B 0,C 180,E1 -16944.772,E2 -16944.772} C_VEL
LIN {X 0,Y 284.551,Z 525.069,A -85,B 0,C 180,E1 -16947.987,E2 -16947.987} C_VEL
LIN {X 0,Y 284.334,Z 524.39,A -85,B 0,C 180,E1 -16951.269,E2 -16951.269} C_VEL
LIN {X 0,Y 284.437,Z 524.724,A -85,B 0,C 180,E1 -16954.631,E2 -16954.631} C_VEL
LIN {X 0,Y 284.866,Z 526.122,A -85,B 0,C 180,E1 -16958.081,E2 -16958.081} C_VEL
LIN {X 0,Y 285.42,Z 527.515,A -85,B 0,C 180,E1 -16960.244,E2 -16960.244} C_VEL
LIN {X 0,Y 286.402,Z 530.434,A -85,B 0,C 180,E1 -16963.4,E2 -16963.4} C_VEL
LIN {X 0,Y 287.962,Z 534.936,A -85,B 0,C 180,E1 -16967.069,E2 -16967.069} C_VEL
LIN {X 0,Y 289.289,Z 539.488,A -85,B 0,C 180,E1 -16969.93,E2 -16969.93} C_VEL
LIN {X 0,Y 290.865,Z 545.003,A -85,B 0,C 180,E1 -16972.879,E2 -16972.879} C_VEL
LIN {X 0,Y 291.517,Z 547.73,A -85,B 0,C 180,E1 -16974.131,E2 -16974.131} C_VEL
LIN {X 0,Y 294.504,Z 553.323,A -85,B 0,C 180,E1 -16975.311,E2 -16975.311} C_VEL
LIN {X 0,Y 296.056,Z 556.304,A -85,B 0,C 180,E1 -16975.891,E2 -16975.891} C_VEL
LIN {X 0,Y 298.725,Z 561.591,A -85,B 0,C 180,E1 -16976.859,E2 -16976.859} C_VEL
LIN {X 0,Y 301.242,Z 567.049,A -85,B 0,C 180,E1 -16977.722,E2 -16977.722} C_VEL
LIN {X 0,Y 302.404,Z 569.847,A -85,B 0,C 180,E1 -16978.126,E2 -16978.126} C_VEL
LIN {X 0,Y 304.799,Z 584.395,A -85,B 0,C 180,E1 -16979.376,E2 -16979.376} C_VEL
LIN {X 0,Y 306.387,Z 599.003,A -85,B 0,C 180,E1 -16980.403,E2 -16980.403} C_VEL
LIN {X 0,Y 306.993,Z 611.516,A -85,B 0,C 180,E1 -16981.122,E2 -16981.122} C_VEL
LIN {X 0,Y 303.155,Z 663.567,A -85,B 0,C 180,E1 -16982.938,E2 -16982.938} C_VEL
LIN {X 0,Y 301.49,Z 676.862,A -85,B 0,C 180,E1 -16983.618,E2 -16983.618} C_VEL
LIN {X 0,Y 299.536,Z 688.858,A -85,B 0,C 180,E1 -16984.461,E2 -16984.461} C_VEL
LIN {X 0,Y 296.925,Z 702.394,A -85,B 0,C 180,E1 -16985.717,E2 -16985.717} C_VEL
LIN {X 0,Y 294.565,Z 713.228,A -85,B 0,C 180,E1 -16987.003,E2 -16987.003} C_VEL
LIN {X 0,Y 292.223,Z 723.226,A -85,B 0,C 180,E1 -16988.484,E2 -16988.484} C_VEL
LIN {X 0,Y 289.875,Z 732.472,A -85,B 0,C 180,E1 -16990.158,E2 -16990.158} C_VEL
LIN {X 0,Y 287.65,Z 741.592,A -85,B 0,C 180,E1 -16992.203,E2 -16992.203} C_VEL
LIN {X 0,Y 286.514,Z 747.175,A -85,B 0,C 180,E1 -16993.616,E2 -16993.616} C_VEL
LIN {X 0,Y 285.032,Z 755.852,A -85,B 0,C 180,E1 -16995.726,E2 -16995.726} C_VEL
LIN {X 0,Y 283.854,Z 762.743,A -85,B 0,C 180,E1 -16997.851,E2 -16997.851} C_VEL
LIN {X 0,Y 283.138,Z 768.252,A -85,B 0,C 180,E1 -16999.994,E2 -16999.994} C_VEL
LIN {X 0,Y 282.683,Z 772.553,A -85,B 0,C 180,E1 -17002.141,E2 -17002.141} C_VEL
LIN {X 0,Y 282.432,Z 776.001,A -85,B 0,C 180,E1 -17004.475,E2 -17004.475} C_VEL
LIN {X 0,Y 282.402,Z 778.535,A -85,B 0,C 180,E1 -17007.147,E2 -17007.147} C_VEL
LIN {X 0,Y 282.367,Z 779.258,A -85,B 0,C 180,E1 -17008.574,E2 -17008.574} C_VEL
LIN {X 0,Y 282.364,Z 779.59,A -85,B 0,C 180,E1 -17010,E2 -17010} C_VEL
LIN {X 0,Y 282.359,Z 779.531,A -85,B 0,C 180,E1 -17011.426,E2 -17011.426} C_VEL
LIN {X 0,Y 282.402,Z 779.059,A -85,B 0,C 180,E1 -17012.853,E2 -17012.853} C_VEL
LIN {X 0,Y 282.441,Z 776.852,A -85,B 0,C 180,E1 -17015.712,E2 -17015.712} C_VEL
LIN {X 0,Y 282.697,Z 774.093,A -85,B 0,C 180,E1 -17017.859,E2 -17017.859} C_VEL
LIN {X 0,Y 283.206,Z 770.303,A -85,B 0,C 180,E1 -17020.003,E2 -17020.003} C_VEL
LIN {X 0,Y 283.981,Z 765.374,A -85,B 0,C 180,E1 -17022.143,E2 -17022.143} C_VEL
LIN {X 0,Y 285.175,Z 759.163,A -85,B 0,C 180,E1 -17024.267,E2 -17024.267} C_VEL
LIN {X 0,Y 286.668,Z 751.38,A -85,B 0,C 180,E1 -17026.375,E2 -17026.375} C_VEL
LIN {X 0,Y 288.179,Z 743.383,A -85,B 0,C 180,E1 -17028.125,E2 -17028.125} C_VEL
LIN {X 0,Y 289.882,Z 733.715,A -85,B 0,C 180,E1 -17029.841,E2 -17029.841} C_VEL
LIN {X 0,Y 291.829,Z 722.853,A -85,B 0,C 180,E1 -17031.361,E2 -17031.361} C_VEL
LIN {X 0,Y 293.407,Z 712.2,A -85,B 0,C 180,E1 -17032.534,E2 -17032.534} C_VEL
LIN {X 0,Y 294.896,Z 700.488,A -85,B 0,C 180,E1 -17033.527,E2 -17033.527} C_VEL
LIN {X 0,Y 296.129,Z 687.873,A -85,B 0,C 180,E1 -17034.306,E2 -17034.306} C_VEL
LIN {X 0,Y 296.981,Z 675.644,A -85,B 0,C 180,E1 -17034.79,E2 -17034.79} C_VEL
LIN {X 0,Y 298.783,Z 608.778,A -85,B 0,C 180,E1 -17036.405,E2 -17036.405} C_VEL
LIN {X 0,Y 294.696,Z 575.84,A -85,B 0,C 180,E1 -17037.703,E2 -17037.703} C_VEL
LIN {X 0,Y 291.996,Z 559.051,A -85,B 0,C 180,E1 -17038.485,E2 -17038.485} C_VEL
LIN {X 0,Y 291.626,Z 552.823,A -85,B 0,C 180,E1 -17039.12,E2 -17039.12} C_VEL
LIN {X 0,Y 287.112,Z 537.43,A -85,B 0,C 180,E1 -17041.116,E2 -17041.116} C_VEL
LIN {X 0,Y 284.387,Z 524.063,A -85,B 0,C 180,E1 -17045.049,E2 -17045.049} C_VEL
LIN {X 0,Y 284.305,Z 524.031,A -85,B 0,C 180,E1 -17048.169,E2 -17048.169} C_VEL
LIN {X 0,Y 284.267,Z 524.077,A -85,B 0,C 180,E1 -17052.124,E2 -17052.124} C_VEL
LIN {X 0,Y 284.286,Z 524.075,A -85,B 0,C 180,E1 -17056.195,E2 -17056.195} C_VEL
LIN {X 0,Y 284.347,Z 524.065,A -85,B 0,C 180,E1 -17060.012,E2 -17060.012} C_VEL
LIN {X 0,Y 284.35,Z 524.05,A -85,B 0,C 180,E1 -17063.617,E2 -17063.617} C_VEL
LIN {X 0,Y 284.303,Z 524.067,A -85,B 0,C 180,E1 -17067.189,E2 -17067.189} C_VEL
LIN {X 0,Y 284.353,Z 524.051,A -85,B 0,C 180,E1 -17070.376,E2 -17070.376} C_VEL
LIN {X 0,Y 284.372,Z 524.057,A -85,B 0,C 180,E1 -17073.586,E2 -17073.586} C_VEL
LIN {X 0,Y 284.327,Z 524.043,A -85,B 0,C 180,E1 -17076.704,E2 -17076.704} C_VEL
LIN {X 0,Y 284.396,Z 524.049,A -85,B 0,C 180,E1 -17081.261,E2 -17081.261} C_VEL
LIN {X 0,Y 284.472,Z 524.026,A -85,B 0,C 180,E1 -17084.47,E2 -17084.47} C_VEL
LIN {X 0,Y 284.483,Z 524.047,A -85,B 0,C 180,E1 -17088.602,E2 -17088.602} C_VEL
LIN {X 0,Y 284.65,Z 523.997,A -85,B 0,C 180,E1 -17091.481,E2 -17091.481} C_VEL
LIN {X 0,Y 284.595,Z 524.028,A -85,B 0,C 180,E1 -17094.331,E2 -17094.331} C_VEL
LIN {X 0,Y 284.85,Z 523.981,A -85,B 0,C 180,E1 -17098.587,E2 -17098.587} C_VEL
LIN {X 0,Y 284.85,Z 523.979,A -85,B 0,C 180,E1 -17101.414,E2 -17101.414} C_VEL
LIN {X 0,Y 284.681,Z 524.001,A -85,B 0,C 180,E1 -17107.091,E2 -17107.091} C_VEL
LIN {X 0,Y 284.513,Z 524.028,A -85,B 0,C 180,E1 -17109.958,E2 -17109.958} C_VEL
LIN {X 0,Y 284.472,Z 524.04,A -85,B 0,C 180,E1 -17114.304,E2 -17114.304} C_VEL
LIN {X 0,Y 284.419,Z 524.034,A -85,B 0,C 180,E1 -17117.249,E2 -17117.249} C_VEL
LIN {X 0,Y 284.374,Z 524.062,A -85,B 0,C 180,E1 -17120.243,E2 -17120.243} C_VEL
LIN {X 0,Y 284.364,Z 524.043,A -85,B 0,C 180,E1 -17123.876,E2 -17123.876} C_VEL
LIN {X 0,Y 284.362,Z 524.058,A -85,B 0,C 180,E1 -17128.008,E2 -17128.008} C_VEL
LIN {X 0,Y 284.295,Z 524.067,A -85,B 0,C 180,E1 -17131.275,E2 -17131.275} C_VEL
LIN {X 0,Y 284.338,Z 524.056,A -85,B 0,C 180,E1 -17135.349,E2 -17135.349} C_VEL
LIN {X 0,Y 284.31,Z 524.073,A -85,B 0,C 180,E1 -17138.17,E2 -17138.17} C_VEL
LIN {X 0,Y 284.268,Z 524.08,A -85,B 0,C 180,E1 -17142.126,E2 -17142.126} C_VEL
LIN {X 0,Y 284.268,Z 524.074,A -85,B 0,C 180,E1 -17146.193,E2 -17146.193} C_VEL
LIN {X 0,Y 284.306,Z 524.067,A -85,B 0,C 180,E1 -17150.025,E2 -17150.025} C_VEL
LIN {X 0,Y 284.319,Z 524.232,A -85,B 0,C 180,E1 -17152.28,E2 -17152.28} C_VEL
LIN {X 0,Y 287.966,Z 536.8,A -85,B 0,C 180,E1 -17155.853,E2 -17155.853} C_VEL
LIN {X 0,Y 290.645,Z 547.533,A -85,B 0,C 180,E1 -17158.677,E2 -17158.677} C_VEL
LIN {X 0,Y 291.408,Z 550.771,A -85,B 0,C 180,E1 -17159.43,E2 -17159.43} C_VEL
LIN {X 0,Y 295.152,Z 560.167,A -85,B 0,C 180,E1 -17160.099,E2 -17160.099} C_VEL
LIN {X 0,Y 299.984,Z 585.957,A -85,B 0,C 180,E1 -17161.294,E2 -17161.294} C_VEL
LIN {X 0,Y 297.685,Z 661.535,A -85,B 0,C 180,E1 -17163.112,E2 -17163.112} C_VEL
LIN {X 0,Y 296.817,Z 674.83,A -85,B 0,C 180,E1 -17163.692,E2 -17163.692} C_VEL
LIN {X 0,Y 295.711,Z 687.04,A -85,B 0,C 180,E1 -17164.504,E2 -17164.504} C_VEL
LIN {X 0,Y 294.362,Z 699.002,A -85,B 0,C 180,E1 -17165.582,E2 -17165.582} C_VEL
LIN {X 0,Y 292.725,Z 709.918,A -85,B 0,C 180,E1 -17166.85,E2 -17166.85} C_VEL
LIN {X 0,Y 290.915,Z 720.333,A -85,B 0,C 180,E1 -17168.383,E2 -17168.383} C_VEL
LIN {X 0,Y 289.075,Z 729.731,A -85,B 0,C 180,E1 -17170.101,E2 -17170.101} C_VEL
LIN {X 0,Y 287.48,Z 737.429,A -85,B 0,C 180,E1 -17171.839,E2 -17171.839} C_VEL
LIN {X 0,Y 286.12,Z 744.457,A -85,B 0,C 180,E1 -17173.801,E2 -17173.801} C_VEL
LIN {X 0,Y 285.065,Z 750.051,A -85,B 0,C 180,E1 -17175.727,E2 -17175.727} C_VEL
LIN {X 0,Y 283.958,Z 754.991,A -85,B 0,C 180,E1 -17177.856,E2 -17177.856} C_VEL
LIN {X 0,Y 283.282,Z 758.793,A -85,B 0,C 180,E1 -17179.999,E2 -17179.999} C_VEL
LIN {X 0,Y 282.92,Z 760.741,A -85,B 0,C 180,E1 -17181.429,E2 -17181.429} C_VEL
LIN {X 0,Y 282.669,Z 762.28,A -85,B 0,C 180,E1 -17182.859,E2 -17182.859} C_VEL
LIN {X 0,Y 282.485,Z 763.446,A -85,B 0,C 180,E1 -17184.372,E2 -17184.372} C_VEL
LIN {X 0,Y 282.397,Z 764.401,A -85,B 0,C 180,E1 -17187.147,E2 -17187.147} C_VEL
LIN {X 0,Y 282.354,Z 764.334,A -85,B 0,C 180,E1 -17188.574,E2 -17188.574} C_VEL
LIN {X 0,Y 282.361,Z 763.85,A -85,B 0,C 180,E1 -17190,E2 -17190} C_VEL
LIN {X 0,Y 282.612,Z 761.68,A -85,B 0,C 180,E1 -17192.851,E2 -17192.851} C_VEL
LIN {X 0,Y 283.04,Z 758.962,A -85,B 0,C 180,E1 -17194.986,E2 -17194.986} C_VEL
LIN {X 0,Y 283.503,Z 755.237,A -85,B 0,C 180,E1 -17197.12,E2 -17197.12} C_VEL
LIN {X 0,Y 284.268,Z 750.394,A -85,B 0,C 180,E1 -17199.247,E2 -17199.247} C_VEL
LIN {X 0,Y 285.313,Z 744.292,A -85,B 0,C 180,E1 -17201.365,E2 -17201.365} C_VEL
LIN {X 0,Y 286.73,Z 736.629,A -85,B 0,C 180,E1 -17203.465,E2 -17203.465} C_VEL
LIN {X 0,Y 288.389,Z 727.078,A -85,B 0,C 180,E1 -17205.549,E2 -17205.549} C_VEL
LIN {X 0,Y 289.949,Z 717.136,A -85,B 0,C 180,E1 -17207.273,E2 -17207.273} C_VEL
LIN {X 0,Y 291.622,Z 705.954,A -85,B 0,C 180,E1 -17208.804,E2 -17208.804} C_VEL
LIN {X 0,Y 292.956,Z 694.994,A -85,B 0,C 180,E1 -17209.99,E2 -17209.99} C_VEL
LIN {X 0,Y 294.206,Z 683.856,A -85,B 0,C 180,E1 -17210.905,E2 -17210.905} C_VEL
LIN {X 0,Y 295.071,Z 670.981,A -85,B 0,C 180,E1 -17211.689,E2 -17211.689} C_VEL
LIN {X 0,Y 295.731,Z 657.456,A -85,B 0,C 180,E1 -17212.209,E2 -17212.209} C_VEL
LIN {X 0,Y 297.699,Z 584.84,A -85,B 0,C 180,E1 -17213.938,E2 -17213.938} C_VEL
LIN {X 0,Y 293.68,Z 561.219,A -85,B 0,C 180,E1 -17214.936,E2 -17214.936} C_VEL
LIN {X 0,Y 291.969,Z 553.685,A -85,B 0,C 180,E1 -17215.304,E2 -17215.304} C_VEL
LIN {X 0,Y 290.761,Z 550.402,A -85,B 0,C 180,E1 -17215.528,E2 -17215.528} C_VEL
LIN {X 0,Y 288.482,Z 539.574,A -85,B 0,C 180,E1 -17218.186,E2 -17218.186} C_VEL
LIN {X 0,Y 285.635,Z 528.67,A -85,B 0,C 180,E1 -17221.11,E2 -17221.11} C_VEL
LIN {X 0,Y 284.316,Z 524.075,A -85,B 0,C 180,E1 -17222.417,E2 -17222.417} C_VEL
LIN {X 0,Y 284.352,Z 524.058,A -85,B 0,C 180,E1 -17226.382,E2 -17226.382} C_VEL
LIN {X 0,Y 284.351,Z 524.055,A -85,B 0,C 180,E1 -17229.986,E2 -17229.986} C_VEL
LIN {X 0,Y 284.317,Z 524.064,A -85,B 0,C 180,E1 -17233.797,E2 -17233.797} C_VEL
LIN {X 0,Y 284.302,Z 524.071,A -85,B 0,C 180,E1 -17238.129,E2 -17238.129} C_VEL
LIN {X 0,Y 284.31,Z 524.097,A -85,B 0,C 180,E1 -17238.846,E2 -17238.846} C_VEL
LIN {X 0,Y 293.578,Z 550.817,A -85,B 0,C 180,E1 -17240.326,E2 -17240.326} C_VEL
LIN {X 0,Y 293.5,Z 553.177,A -85,B 0,C 180,E1 -17240.403,E2 -17240.403} C_VEL
LIN {X 0,Y 292.694,Z 558.97,A -85,B 0,C 180,E1 -17240.557,E2 -17240.557} C_VEL
LIN {X 0,Y 286.454,Z 577.743,A -85,B 0,C 180,E1 -17240.866,E2 -17240.866} C_VEL
LIN {X 0,Y 285.48,Z 583.539,A -85,B 0,C 180,E1 -17241.017,E2 -17241.017} C_VEL
LIN {X 0,Y 284.106,Z 624.847,A -85,B 0,C 180,E1 -17242.422,E2 -17242.422} C_VEL
LIN {X 0,Y 283.461,Z 638.684,A -85,B 0,C 180,E1 -17243.187,E2 -17243.187} C_VEL
LIN {X 0,Y 282.531,Z 651.835,A -85,B 0,C 180,E1 -17244.227,E2 -17244.227} C_VEL
LIN {X 0,Y 281.484,Z 664.798,A -85,B 0,C 180,E1 -17245.581,E2 -17245.581} C_VEL
LIN {X 0,Y 280.303,Z 676.584,A -85,B 0,C 180,E1 -17247.166,E2 -17247.166} C_VEL
LIN {X 0,Y 279.338,Z 686.435,A -85,B 0,C 180,E1 -17248.804,E2 -17248.804} C_VEL
LIN {X 0,Y 278.355,Z 694.883,A -85,B 0,C 180,E1 -17250.505,E2 -17250.505} C_VEL
LIN {X 0,Y 277.506,Z 702.715,A -85,B 0,C 180,E1 -17252.421,E2 -17252.421} C_VEL
LIN {X 0,Y 276.764,Z 710.618,A -85,B 0,C 180,E1 -17254.827,E2 -17254.827} C_VEL
LIN {X 0,Y 276.261,Z 716.028,A -85,B 0,C 180,E1 -17256.897,E2 -17256.897} C_VEL
LIN {X 0,Y 275.871,Z 720.577,A -85,B 0,C 180,E1 -17259.104,E2 -17259.104} C_VEL
LIN {X 0,Y 275.735,Z 723.059,A -85,B 0,C 180,E1 -17260.649,E2 -17260.649} C_VEL
LIN {X 0,Y 275.647,Z 725.022,A -85,B 0,C 180,E1 -17262.184,E2 -17262.184} C_VEL
LIN {X 0,Y 275.637,Z 726.516,A -85,B 0,C 180,E1 -17263.711,E2 -17263.711} C_VEL
LIN {X 0,Y 275.816,Z 727.622,A -85,B 0,C 180,E1 -17265.522,E2 -17265.522} C_VEL
LIN {X 0,Y 276.294,Z 728.13,A -85,B 0,C 180,E1 -17268.258,E2 -17268.258} C_VEL
LIN {X 0,Y 276.708,Z 727.748,A -85,B 0,C 180,E1 -17269.759,E2 -17269.759} C_VEL
LIN {X 0,Y 277.281,Z 726.907,A -85,B 0,C 180,E1 -17271.293,E2 -17271.293} C_VEL
LIN {X 0,Y 277.853,Z 725.715,A -85,B 0,C 180,E1 -17272.734,E2 -17272.734} C_VEL
LIN {X 0,Y 279.01,Z 722.984,A -85,B 0,C 180,E1 -17274.942,E2 -17274.942} C_VEL
LIN {X 0,Y 280.482,Z 719.179,A -85,B 0,C 180,E1 -17277.127,E2 -17277.127} C_VEL
LIN {X 0,Y 282.211,Z 714.226,A -85,B 0,C 180,E1 -17279.286,E2 -17279.286} C_VEL
LIN {X 0,Y 284.196,Z 707.952,A -85,B 0,C 180,E1 -17281.417,E2 -17281.417} C_VEL
LIN {X 0,Y 286.628,Z 700.058,A -85,B 0,C 180,E1 -17283.514,E2 -17283.514} C_VEL
LIN {X 0,Y 288.84,Z 692.085,A -85,B 0,C 180,E1 -17285.235,E2 -17285.235} C_VEL
LIN {X 0,Y 290.758,Z 684.272,A -85,B 0,C 180,E1 -17286.639,E2 -17286.639} C_VEL
LIN {X 0,Y 293.057,Z 674.291,A -85,B 0,C 180,E1 -17288.099,E2 -17288.099} C_VEL
LIN {X 0,Y 295.294,Z 662.91,A -85,B 0,C 180,E1 -17289.417,E2 -17289.417} C_VEL
LIN {X 0,Y 297.223,Z 650.438,A -85,B 0,C 180,E1 -17290.559,E2 -17290.559} C_VEL
LIN {X 0,Y 298.839,Z 636.757,A -85,B 0,C 180,E1 -17291.488,E2 -17291.488} C_VEL
LIN {X 0,Y 299.981,Z 623.76,A -85,B 0,C 180,E1 -17292.086,E2 -17292.086} C_VEL
LIN {X 0,Y 304.561,Z 567.6,A -85,B 0,C 180,E1 -17294.095,E2 -17294.095} C_VEL
LIN {X 0,Y 299.172,Z 557.477,A -85,B 0,C 180,E1 -17295.829,E2 -17295.829} C_VEL
LIN {X 0,Y 294.605,Z 550.235,A -85,B 0,C 180,E1 -17297.407,E2 -17297.407} C_VEL
LIN {X 0,Y 291.569,Z 545.914,A -85,B 0,C 180,E1 -17298.524,E2 -17298.524} C_VEL
LIN {X 0,Y 289.066,Z 542.592,A -85,B 0,C 180,E1 -17299.518,E2 -17299.518} C_VEL
LIN {X 0,Y 286.446,Z 539.117,A -85,B 0,C 180,E1 -17300.638,E2 -17300.638} C_VEL
LIN {X 0,Y 282.926,Z 534.87,A -85,B 0,C 180,E1 -17302.289,E2 -17302.289} C_VEL
LIN {X 0,Y 279.988,Z 531.774,A -85,B 0,C 180,E1 -17303.854,E2 -17303.854} C_VEL
LIN {X 0,Y 279.207,Z 530.439,A -85,B 0,C 180,E1 -17304.392,E2 -17304.392} C_VEL
LIN {X 0,Y 278.466,Z 528.641,A -85,B 0,C 180,E1 -17308.654,E2 -17308.654} C_VEL
LIN {X 0,Y 278.372,Z 528.255,A -85,B 0,C 180,E1 -17312.018,E2 -17312.018} C_VEL
LIN {X 0,Y 278.545,Z 528.828,A -85,B 0,C 180,E1 -17315.473,E2 -17315.473} C_VEL
LIN {X 0,Y 279.174,Z 530.524,A -85,B 0,C 180,E1 -17319.002,E2 -17319.002} C_VEL
LIN {X 0,Y 280.126,Z 533.421,A -85,B 0,C 180,E1 -17322.64,E2 -17322.64} C_VEL
LIN {X 0,Y 281.586,Z 537.698,A -85,B 0,C 180,E1 -17326.369,E2 -17326.369} C_VEL
LIN {X 0,Y 283.079,Z 542.827,A -85,B 0,C 180,E1 -17329.798,E2 -17329.798} C_VEL
LIN {X 0,Y 284.171,Z 546.332,A -85,B 0,C 180,E1 -17331.687,E2 -17331.687} C_VEL
LIN {X 0,Y 287.594,Z 552.432,A -85,B 0,C 180,E1 -17333.29,E2 -17333.29} C_VEL
LIN {X 0,Y 289.095,Z 555.286,A -85,B 0,C 180,E1 -17333.943,E2 -17333.943} C_VEL
LIN {X 0,Y 292.104,Z 560.896,A -85,B 0,C 180,E1 -17335.168,E2 -17335.168} C_VEL
LIN {X 0,Y 295.177,Z 567.349,A -85,B 0,C 180,E1 -17336.357,E2 -17336.357} C_VEL
LIN {X 0,Y 297.794,Z 573.42,A -85,B 0,C 180,E1 -17337.329,E2 -17337.329} C_VEL
LIN {X 0,Y 299.865,Z 586.874,A -85,B 0,C 180,E1 -17338.53,E2 -17338.53} C_VEL
LIN {X 0,Y 301.253,Z 601.096,A -85,B 0,C 180,E1 -17339.562,E2 -17339.562} C_VEL
LIN {X 0,Y 301.741,Z 612.617,A -85,B 0,C 180,E1 -17340.238,E2 -17340.238} C_VEL
LIN {X 0,Y 297.693,Z 663.1,A -85,B 0,C 180,E1 -17342.065,E2 -17342.065} C_VEL
LIN {X 0,Y 295.843,Z 676.95,A -85,B 0,C 180,E1 -17342.788,E2 -17342.788} C_VEL
LIN {X 0,Y 293.639,Z 689.659,A -85,B 0,C 180,E1 -17343.719,E2 -17343.719} C_VEL
LIN {X 0,Y 290.897,Z 702.836,A -85,B 0,C 180,E1 -17344.989,E2 -17344.989} C_VEL
LIN {X 0,Y 288.139,Z 714.499,A -85,B 0,C 180,E1 -17346.46,E2 -17346.46} C_VEL
LIN {X 0,Y 285.194,Z 726.109,A -85,B 0,C 180,E1 -17348.307,E2 -17348.307} C_VEL
LIN {X 0,Y 282.86,Z 734.768,A -85,B 0,C 180,E1 -17350.024,E2 -17350.024} C_VEL
LIN {X 0,Y 280.543,Z 743.481,A -85,B 0,C 180,E1 -17352.167,E2 -17352.167} C_VEL
LIN {X 0,Y 279.381,Z 748.505,A -85,B 0,C 180,E1 -17353.561,E2 -17353.561} C_VEL
LIN {X 0,Y 277.883,Z 756.821,A -85,B 0,C 180,E1 -17355.725,E2 -17355.725} C_VEL
LIN {X 0,Y 276.721,Z 763.5,A -85,B 0,C 180,E1 -17357.906,E2 -17357.906} C_VEL
LIN {X 0,Y 275.921,Z 769.597,A -85,B 0,C 180,E1 -17360.47,E2 -17360.47} C_VEL
LIN {X 0,Y 275.515,Z 773.532,A -85,B 0,C 180,E1 -17362.673,E2 -17362.673} C_VEL
LIN {X 0,Y 275.354,Z 776.003,A -85,B 0,C 180,E1 -17364.513,E2 -17364.513} C_VEL
LIN {X 0,Y 275.308,Z 778.33,A -85,B 0,C 180,E1 -17367.074,E2 -17367.074} C_VEL
LIN {X 0,Y 275.291,Z 779.06,A -85,B 0,C 180,E1 -17368.537,E2 -17368.537} C_VEL
LIN {X 0,Y 275.285,Z 779.397,A -85,B 0,C 180,E1 -17370,E2 -17370} C_VEL
LIN {X 0,Y 275.284,Z 779.343,A -85,B 0,C 180,E1 -17371.463,E2 -17371.463} C_VEL
LIN {X 0,Y 275.308,Z 778.88,A -85,B 0,C 180,E1 -17372.926,E2 -17372.926} C_VEL
LIN {X 0,Y 275.349,Z 776.683,A -85,B 0,C 180,E1 -17375.86,E2 -17375.86} C_VEL
LIN {X 0,Y 275.65,Z 773.934,A -85,B 0,C 180,E1 -17378.061,E2 -17378.061} C_VEL
LIN {X 0,Y 276.189,Z 770.156,A -85,B 0,C 180,E1 -17380.26,E2 -17380.26} C_VEL
LIN {X 0,Y 276.994,Z 765.239,A -85,B 0,C 180,E1 -17382.454,E2 -17382.454} C_VEL
LIN {X 0,Y 278.279,Z 759.043,A -85,B 0,C 180,E1 -17384.628,E2 -17384.628} C_VEL
LIN {X 0,Y 279.855,Z 751.284,A -85,B 0,C 180,E1 -17386.786,E2 -17386.786} C_VEL
LIN {X 0,Y 281.541,Z 742.636,A -85,B 0,C 180,E1 -17388.711,E2 -17388.711} C_VEL
LIN {X 0,Y 283.433,Z 732.602,A -85,B 0,C 180,E1 -17390.502,E2 -17390.502} C_VEL
LIN {X 0,Y 285.454,Z 721.44,A -85,B 0,C 180,E1 -17392.052,E2 -17392.052} C_VEL
LIN {X 0,Y 287.108,Z 710.503,A -85,B 0,C 180,E1 -17393.248,E2 -17393.248} C_VEL
LIN {X 0,Y 288.702,Z 698.362,A -85,B 0,C 180,E1 -17394.254,E2 -17394.254} C_VEL
LIN {X 0,Y 289.916,Z 685.526,A -85,B 0,C 180,E1 -17395.005,E2 -17395.005} C_VEL
LIN {X 0,Y 290.715,Z 671.974,A -85,B 0,C 180,E1 -17395.506,E2 -17395.506} C_VEL
LIN {X 0,Y 292.451,Z 609.507,A -85,B 0,C 180,E1 -17397.025,E2 -17397.025} C_VEL
LIN {X 0,Y 288.478,Z 576.908,A -85,B 0,C 180,E1 -17398.346,E2 -17398.346} C_VEL
LIN {X 0,Y 285.563,Z 558.93,A -85,B 0,C 180,E1 -17399.212,E2 -17399.212} C_VEL
LIN {X 0,Y 285.217,Z 554.458,A -85,B 0,C 180,E1 -17399.705,E2 -17399.705} C_VEL
LIN {X 0,Y 280.32,Z 538.261,A -85,B 0,C 180,E1 -17401.916,E2 -17401.916} C_VEL
LIN {X 0,Y 279.236,Z 534.346,A -85,B 0,C 180,E1 -17402.491,E2 -17402.491} C_VEL
LIN {X 0,Y 277.333,Z 524.938,A -85,B 0,C 180,E1 -17405.372,E2 -17405.372} C_VEL
LIN {X 0,Y 277.23,Z 524.919,A -85,B 0,C 180,E1 -17409.328,E2 -17409.328} C_VEL
LIN {X 0,Y 277.213,Z 524.946,A -85,B 0,C 180,E1 -17413.196,E2 -17413.196} C_VEL
LIN {X 0,Y 277.237,Z 524.943,A -85,B 0,C 180,E1 -17417.319,E2 -17417.319} C_VEL
LIN {X 0,Y 277.263,Z 524.949,A -85,B 0,C 180,E1 -17420.677,E2 -17420.677} C_VEL
LIN {X 0,Y 277.301,Z 524.931,A -85,B 0,C 180,E1 -17424.344,E2 -17424.344} C_VEL
LIN {X 0,Y 277.239,Z 524.942,A -85,B 0,C 180,E1 -17427.836,E2 -17427.836} C_VEL
LIN {X 0,Y 277.284,Z 524.938,A -85,B 0,C 180,E1 -17431.212,E2 -17431.212} C_VEL
LIN {X 0,Y 277.304,Z 524.928,A -85,B 0,C 180,E1 -17434.479,E2 -17434.479} C_VEL
LIN {X 0,Y 277.262,Z 524.933,A -85,B 0,C 180,E1 -17437.653,E2 -17437.653} C_VEL
LIN {X 0,Y 277.338,Z 524.934,A -85,B 0,C 180,E1 -17440.766,E2 -17440.766} C_VEL
LIN {X 0,Y 277.422,Z 524.912,A -85,B 0,C 180,E1 -17445.325,E2 -17445.325} C_VEL
LIN {X 0,Y 277.501,Z 524.905,A -85,B 0,C 180,E1 -17449.789,E2 -17449.789} C_VEL
LIN {X 0,Y 277.644,Z 524.875,A -85,B 0,C 180,E1 -17452.729,E2 -17452.729} C_VEL
LIN {X 0,Y 277.816,Z 524.857,A -85,B 0,C 180,E1 -17458.551,E2 -17458.551} C_VEL
LIN {X 0,Y 277.816,Z 524.854,A -85,B 0,C 180,E1 -17461.45,E2 -17461.45} C_VEL
LIN {X 0,Y 277.636,Z 524.877,A -85,B 0,C 180,E1 -17467.272,E2 -17467.272} C_VEL
LIN {X 0,Y 277.455,Z 524.91,A -85,B 0,C 180,E1 -17470.214,E2 -17470.214} C_VEL
LIN {X 0,Y 277.423,Z 524.911,A -85,B 0,C 180,E1 -17474.675,E2 -17474.675} C_VEL
LIN {X 0,Y 277.34,Z 524.938,A -85,B 0,C 180,E1 -17479.235,E2 -17479.235} C_VEL
LIN {X 0,Y 277.315,Z 524.923,A -85,B 0,C 180,E1 -17484.171,E2 -17484.171} C_VEL
LIN {X 0,Y 277.333,Z 524.935,A -85,B 0,C 180,E1 -17487.51,E2 -17487.51} C_VEL
LIN {X 0,Y 277.269,Z 524.934,A -85,B 0,C 180,E1 -17490.482,E2 -17490.482} C_VEL
LIN {X 0,Y 277.244,Z 524.943,A -85,B 0,C 180,E1 -17493.897,E2 -17493.897} C_VEL
LIN {X 0,Y 277.265,Z 524.952,A -85,B 0,C 180,E1 -17497.47,E2 -17497.47} C_VEL
LIN {X 0,Y 277.208,Z 524.959,A -85,B 0,C 180,E1 -17501.238,E2 -17501.238} C_VEL
LIN {X 0,Y 277.216,Z 524.959,A -85,B 0,C 180,E1 -17505.224,E2 -17505.224} C_VEL
LIN {X 0,Y 277.222,Z 524.949,A -85,B 0,C 180,E1 -17509.513,E2 -17509.513} C_VEL
LIN {X 0,Y 277.264,Z 525.082,A -85,B 0,C 180,E1 -17511.453,E2 -17511.453} C_VEL
LIN {X 0,Y 280.74,Z 536.673,A -85,B 0,C 180,E1 -17514.847,E2 -17514.847} C_VEL
LIN {X 0,Y 283.634,Z 548.159,A -85,B 0,C 180,E1 -17517.964,E2 -17517.964} C_VEL
LIN {X 0,Y 284.354,Z 550.994,A -85,B 0,C 180,E1 -17518.627,E2 -17518.627} C_VEL
LIN {X 0,Y 289.19,Z 562.566,A -85,B 0,C 180,E1 -17519.512,E2 -17519.512} C_VEL
LIN {X 0,Y 293.701,Z 586.865,A -85,B 0,C 180,E1 -17520.673,E2 -17520.673} C_VEL
LIN {X 0,Y 291.285,Z 662.161,A -85,B 0,C 180,E1 -17522.521,E2 -17522.521} C_VEL
LIN {X 0,Y 290.393,Z 675.254,A -85,B 0,C 180,E1 -17523.111,E2 -17523.111} C_VEL
LIN {X 0,Y 289.223,Z 687.734,A -85,B 0,C 180,E1 -17523.966,E2 -17523.966} C_VEL
LIN {X 0,Y 287.844,Z 699.243,A -85,B 0,C 180,E1 -17525.029,E2 -17525.029} C_VEL
LIN {X 0,Y 286.199,Z 709.906,A -85,B 0,C 180,E1 -17526.29,E2 -17526.29} C_VEL
LIN {X 0,Y 284.321,Z 720.357,A -85,B 0,C 180,E1 -17527.855,E2 -17527.855} C_VEL
LIN {X 0,Y 282.385,Z 729.784,A -85,B 0,C 180,E1 -17529.609,E2 -17529.609} C_VEL
LIN {X 0,Y 280.718,Z 737.505,A -85,B 0,C 180,E1 -17531.386,E2 -17531.386} C_VEL
LIN {X 0,Y 279.227,Z 744.768,A -85,B 0,C 180,E1 -17533.46,E2 -17533.46} C_VEL
LIN {X 0,Y 278.159,Z 750.172,A -85,B 0,C 180,E1 -17535.365,E2 -17535.365} C_VEL
LIN {X 0,Y 276.993,Z 755.128,A -85,B 0,C 180,E1 -17537.546,E2 -17537.546} C_VEL
LIN {X 0,Y 276.25,Z 758.944,A -85,B 0,C 180,E1 -17539.742,E2 -17539.742} C_VEL
LIN {X 0,Y 275.892,Z 760.898,A -85,B 0,C 180,E1 -17541.209,E2 -17541.209} C_VEL
LIN {X 0,Y 275.607,Z 762.444,A -85,B 0,C 180,E1 -17542.675,E2 -17542.675} C_VEL
LIN {X 0,Y 275.377,Z 763.752,A -85,B 0,C 180,E1 -17544.47,E2 -17544.47} C_VEL
LIN {X 0,Y 275.306,Z 764.589,A -85,B 0,C 180,E1 -17547.074,E2 -17547.074} C_VEL
LIN {X 0,Y 275.279,Z 764.527,A -85,B 0,C 180,E1 -17548.537,E2 -17548.537} C_VEL
LIN {X 0,Y 275.283,Z 764.056,A -85,B 0,C 180,E1 -17550,E2 -17550} C_VEL
LIN {X 0,Y 275.546,Z 761.898,A -85,B 0,C 180,E1 -17552.924,E2 -17552.924} C_VEL
LIN {X 0,Y 275.973,Z 759.192,A -85,B 0,C 180,E1 -17555.114,E2 -17555.114} C_VEL
LIN {X 0,Y 276.635,Z 754.561,A -85,B 0,C 180,E1 -17557.77,E2 -17557.77} C_VEL
LIN {X 0,Y 277.616,Z 748.759,A -85,B 0,C 180,E1 -17560.207,E2 -17560.207} C_VEL
LIN {X 0,Y 278.801,Z 742.188,A -85,B 0,C 180,E1 -17562.372,E2 -17562.372} C_VEL
LIN {X 0,Y 280.382,Z 734.005,A -85,B 0,C 180,E1 -17564.516,E2 -17564.516} C_VEL
LIN {X 0,Y 281.9,Z 725.568,A -85,B 0,C 180,E1 -17566.288,E2 -17566.288} C_VEL
LIN {X 0,Y 283.389,Z 716.355,A -85,B 0,C 180,E1 -17567.872,E2 -17567.872} C_VEL
LIN {X 0,Y 284.937,Z 706.34,A -85,B 0,C 180,E1 -17569.262,E2 -17569.262} C_VEL
LIN {X 0,Y 286.318,Z 695.426,A -85,B 0,C 180,E1 -17570.474,E2 -17570.474} C_VEL
LIN {X 0,Y 287.617,Z 684.386,A -85,B 0,C 180,E1 -17571.407,E2 -17571.407} C_VEL
LIN {X 0,Y 288.536,Z 671.209,A -85,B 0,C 180,E1 -17572.23,E2 -17572.23} C_VEL
LIN {X 0,Y 289.186,Z 658.654,A -85,B 0,C 180,E1 -17572.732,E2 -17572.732} C_VEL
LIN {X 0,Y 291.284,Z 585.978,A -85,B 0,C 180,E1 -17574.5,E2 -17574.5} C_VEL
LIN {X 0,Y 287.389,Z 562.746,A -85,B 0,C 180,E1 -17575.51,E2 -17575.51} C_VEL
LIN {X 0,Y 285.957,Z 556.353,A -85,B 0,C 180,E1 -17575.83,E2 -17575.83} C_VEL
LIN {X 0,Y 283.694,Z 550.48,A -85,B 0,C 180,E1 -17576.251,E2 -17576.251} C_VEL
LIN {X 0,Y 281.283,Z 539.584,A -85,B 0,C 180,E1 -17579.014,E2 -17579.014} C_VEL
LIN {X 0,Y 278.328,Z 528.695,A -85,B 0,C 180,E1 -17582.023,E2 -17582.023} C_VEL
LIN {X 0,Y 277.253,Z 524.947,A -85,B 0,C 180,E1 -17583.099,E2 -17583.099} C_VEL
LIN {X 0,Y 277.326,Z 524.936,A -85,B 0,C 180,E1 -17585.811,E2 -17585.811} C_VEL
LIN {X 0,Y 277.266,Z 524.942,A -85,B 0,C 180,E1 -17589.322,E2 -17589.322} C_VEL
LIN {X 0,Y 277.262,Z 524.947,A -85,B 0,C 180,E1 -17593.186,E2 -17593.186} C_VEL
LIN {X 0,Y 277.231,Z 524.952,A -85,B 0,C 180,E1 -17597.32,E2 -17597.32} C_VEL
LIN {X 0,Y 277.302,Z 525.057,A -85,B 0,C 180,E1 -17598.44,E2 -17598.44} C_VEL
LIN {X 0,Y 286.596,Z 551.432,A -85,B 0,C 180,E1 -17599.955,E2 -17599.955} C_VEL
LIN {X 0,Y 285.48,Z 583.539,A -85,B 0,C 180,E1 -17601.017,E2 -17601.017} C_VEL
LIN {X 0,Y 284.52,Z 589.327,A -85,B 0,C 180,E1 -17601.168,E2 -17601.168} C_VEL
LIN {X 0,Y 278.392,Z 608.092,A -85,B 0,C 180,E1 -17601.525,E2 -17601.525} C_VEL
LIN {X 0,Y 277.544,Z 613.877,A -85,B 0,C 180,E1 -17601.694,E2 -17601.694} C_VEL
LIN {X 0,Y 276.938,Z 629.409,A -85,B 0,C 180,E1 -17602.332,E2 -17602.332} C_VEL
LIN {X 0,Y 276.174,Z 643.901,A -85,B 0,C 180,E1 -17603.271,E2 -17603.271} C_VEL
LIN {X 0,Y 275.269,Z 655.997,A -85,B 0,C 180,E1 -17604.345,E2 -17604.345} C_VEL
LIN {X 0,Y 274.054,Z 669.236,A -85,B 0,C 180,E1 -17605.876,E2 -17605.876} C_VEL
LIN {X 0,Y 272.894,Z 680.716,A -85,B 0,C 180,E1 -17607.58,E2 -17607.58} C_VEL
LIN {X 0,Y 271.869,Z 690.125,A -85,B 0,C 180,E1 -17609.299,E2 -17609.299} C_VEL
LIN {X 0,Y 270.851,Z 699.499,A -85,B 0,C 180,E1 -17611.396,E2 -17611.396} C_VEL
LIN {X 0,Y 269.972,Z 707.808,A -85,B 0,C 180,E1 -17613.733,E2 -17613.733} C_VEL
LIN {X 0,Y 269.391,Z 714.09,A -85,B 0,C 180,E1 -17615.934,E2 -17615.934} C_VEL
LIN {X 0,Y 268.863,Z 719.863,A -85,B 0,C 180,E1 -17618.533,E2 -17618.533} C_VEL
LIN {X 0,Y 268.665,Z 722.94,A -85,B 0,C 180,E1 -17620.339,E2 -17620.339} C_VEL
LIN {X 0,Y 268.58,Z 724.813,A -85,B 0,C 180,E1 -17621.699,E2 -17621.699} C_VEL
LIN {X 0,Y 268.537,Z 726.48,A -85,B 0,C 180,E1 -17623.268,E2 -17623.268} C_VEL
LIN {X 0,Y 268.729,Z 728.02,A -85,B 0,C 180,E1 -17625.381,E2 -17625.381} C_VEL
LIN {X 0,Y 269.138,Z 728.747,A -85,B 0,C 180,E1 -17627.941,E2 -17627.941} C_VEL
LIN {X 0,Y 269.557,Z 728.599,A -85,B 0,C 180,E1 -17629.484,E2 -17629.484} C_VEL
LIN {X 0,Y 270.192,Z 727.866,A -85,B 0,C 180,E1 -17631.264,E2 -17631.264} C_VEL
LIN {X 0,Y 271.464,Z 725.49,A -85,B 0,C 180,E1 -17634.056,E2 -17634.056} C_VEL
LIN {X 0,Y 272.873,Z 722.406,A -85,B 0,C 180,E1 -17636.308,E2 -17636.308} C_VEL
LIN {X 0,Y 274.549,Z 718.224,A -85,B 0,C 180,E1 -17638.533,E2 -17638.533} C_VEL
LIN {X 0,Y 276.516,Z 712.835,A -85,B 0,C 180,E1 -17640.728,E2 -17640.728} C_VEL
LIN {X 0,Y 278.831,Z 706.073,A -85,B 0,C 180,E1 -17642.889,E2 -17642.889} C_VEL
LIN {X 0,Y 281.533,Z 697.608,A -85,B 0,C 180,E1 -17645.012,E2 -17645.012} C_VEL
LIN {X 0,Y 284.088,Z 688.363,A -85,B 0,C 180,E1 -17646.878,E2 -17646.878} C_VEL
LIN {X 0,Y 286.881,Z 677.224,A -85,B 0,C 180,E1 -17648.63,E2 -17648.63} C_VEL
LIN {X 0,Y 289.233,Z 666.602,A -85,B 0,C 180,E1 -17649.97,E2 -17649.97} C_VEL
LIN {X 0,Y 291.291,Z 655.014,A -85,B 0,C 180,E1 -17651.129,E2 -17651.129} C_VEL
LIN {X 0,Y 293.225,Z 640.933,A -85,B 0,C 180,E1 -17652.193,E2 -17652.193} C_VEL
LIN {X 0,Y 294.531,Z 627.59,A -85,B 0,C 180,E1 -17652.883,E2 -17652.883} C_VEL
LIN {X 0,Y 298.87,Z 577.908,A -85,B 0,C 180,E1 -17654.721,E2 -17654.721} C_VEL
LIN {X 0,Y 299.492,Z 570.448,A -85,B 0,C 180,E1 -17655.013,E2 -17655.013} C_VEL
LIN {X 0,Y 295.007,Z 562.028,A -85,B 0,C 180,E1 -17656.549,E2 -17656.549} C_VEL
LIN {X 0,Y 291.06,Z 555.64,A -85,B 0,C 180,E1 -17657.988,E2 -17657.988} C_VEL
LIN {X 0,Y 286.923,Z 549.528,A -85,B 0,C 180,E1 -17659.664,E2 -17659.664} C_VEL
LIN {X 0,Y 283.722,Z 545.325,A -85,B 0,C 180,E1 -17661.087,E2 -17661.087} C_VEL
LIN {X 0,Y 280.431,Z 541.237,A -85,B 0,C 180,E1 -17662.715,E2 -17662.715} C_VEL
LIN {X 0,Y 277.375,Z 537.766,A -85,B 0,C 180,E1 -17664.443,E2 -17664.443} C_VEL
LIN {X 0,Y 276.728,Z 536.918,A -85,B 0,C 180,E1 -17664.866,E2 -17664.866} C_VEL
LIN {X 0,Y 273.438,Z 533.937,A -85,B 0,C 180,E1 -17667.143,E2 -17667.143} C_VEL
LIN {X 0,Y 272.562,Z 532.608,A -85,B 0,C 180,E1 -17668.07,E2 -17668.07} C_VEL
LIN {X 0,Y 272.403,Z 532.088,A -85,B 0,C 180,E1 -17671.638,E2 -17671.638} C_VEL
LIN {X 0,Y 272.49,Z 532.482,A -85,B 0,C 180,E1 -17674.57,E2 -17674.57} C_VEL
LIN {X 0,Y 272.973,Z 533.883,A -85,B 0,C 180,E1 -17678.163,E2 -17678.163} C_VEL
LIN {X 0,Y 273.899,Z 536.6,A -85,B 0,C 180,E1 -17681.918,E2 -17681.918} C_VEL
LIN {X 0,Y 275.229,Z 540.477,A -85,B 0,C 180,E1 -17685.642,E2 -17685.642} C_VEL
LIN {X 0,Y 276.362,Z 544.194,A -85,B 0,C 180,E1 -17688.285,E2 -17688.285} C_VEL
LIN {X 0,Y 280.24,Z 550.851,A -85,B 0,C 180,E1 -17690.624,E2 -17690.624} C_VEL
LIN {X 0,Y 281.449,Z 552.653,A -85,B 0,C 180,E1 -17691.227,E2 -17691.227} C_VEL
LIN {X 0,Y 285.332,Z 559.82,A -85,B 0,C 180,E1 -17693.132,E2 -17693.132} C_VEL
LIN {X 0,Y 288.469,Z 566.074,A -85,B 0,C 180,E1 -17694.523,E2 -17694.523} C_VEL
LIN {X 0,Y 291.974,Z 573.726,A -85,B 0,C 180,E1 -17695.957,E2 -17695.957} C_VEL
LIN {X 0,Y 293.525,Z 577.957,A -85,B 0,C 180,E1 -17696.609,E2 -17696.609} C_VEL
LIN {X 0,Y 295.275,Z 591.413,A -85,B 0,C 180,E1 -17697.804,E2 -17697.804} C_VEL
LIN {X 0,Y 296.377,Z 604.516,A -85,B 0,C 180,E1 -17698.776,E2 -17698.776} C_VEL
LIN {X 0,Y 296.541,Z 614.259,A -85,B 0,C 180,E1 -17699.346,E2 -17699.346} C_VEL
LIN {X 0,Y 292.524,Z 661.762,A -85,B 0,C 180,E1 -17701.091,E2 -17701.091} C_VEL
LIN {X 0,Y 290.473,Z 676.135,A -85,B 0,C 180,E1 -17701.849,E2 -17701.849} C_VEL
LIN {X 0,Y 288.159,Z 688.709,A -85,B 0,C 180,E1 -17702.788,E2 -17702.788} C_VEL
LIN {X 0,Y 285.267,Z 701.875,A -85,B 0,C 180,E1 -17704.069,E2 -17704.069} C_VEL
LIN {X 0,Y 282.315,Z 713.613,A -85,B 0,C 180,E1 -17705.553,E2 -17705.553} C_VEL
LIN {X 0,Y 279.748,Z 723.268,A -85,B 0,C 180,E1 -17707.083,E2 -17707.083} C_VEL
LIN {X 0,Y 277.107,Z 732.249,A -85,B 0,C 180,E1 -17708.814,E2 -17708.814} C_VEL
LIN {X 0,Y 274.564,Z 741.278,A -85,B 0,C 180,E1 -17710.991,E2 -17710.991} C_VEL
LIN {X 0,Y 272.244,Z 749.711,A -85,B 0,C 180,E1 -17713.503,E2 -17713.503} C_VEL
LIN {X 0,Y 270.747,Z 757.786,A -85,B 0,C 180,E1 -17715.724,E2 -17715.724} C_VEL
LIN {X 0,Y 269.583,Z 764.251,A -85,B 0,C 180,E1 -17717.962,E2 -17717.962} C_VEL
LIN {X 0,Y 268.888,Z 769.363,A -85,B 0,C 180,E1 -17720.219,E2 -17720.219} C_VEL
LIN {X 0,Y 268.448,Z 773.308,A -85,B 0,C 180,E1 -17722.479,E2 -17722.479} C_VEL
LIN {X 0,Y 268.265,Z 776.031,A -85,B 0,C 180,E1 -17724.576,E2 -17724.576} C_VEL
LIN {X 0,Y 268.217,Z 778.125,A -85,B 0,C 180,E1 -17726.996,E2 -17726.996} C_VEL
LIN {X 0,Y 268.217,Z 778.862,A -85,B 0,C 180,E1 -17728.499,E2 -17728.499} C_VEL
LIN {X 0,Y 268.209,Z 779.204,A -85,B 0,C 180,E1 -17730,E2 -17730} C_VEL
LIN {X 0,Y 268.21,Z 779.155,A -85,B 0,C 180,E1 -17731.501,E2 -17731.501} C_VEL
LIN {X 0,Y 268.217,Z 778.7,A -85,B 0,C 180,E1 -17733.004,E2 -17733.004} C_VEL
LIN {X 0,Y 268.286,Z 776.514,A -85,B 0,C 180,E1 -17736.015,E2 -17736.015} C_VEL
LIN {X 0,Y 268.589,Z 773.776,A -85,B 0,C 180,E1 -17738.274,E2 -17738.274} C_VEL
LIN {X 0,Y 269.187,Z 770.009,A -85,B 0,C 180,E1 -17740.53,E2 -17740.53} C_VEL
LIN {X 0,Y 270.029,Z 765.105,A -85,B 0,C 180,E1 -17742.781,E2 -17742.781} C_VEL
LIN {X 0,Y 271.402,Z 758.923,A -85,B 0,C 180,E1 -17745.007,E2 -17745.007} C_VEL
LIN {X 0,Y 273.062,Z 751.189,A -85,B 0,C 180,E1 -17747.216,E2 -17747.216} C_VEL
LIN {X 0,Y 275.009,Z 741.508,A -85,B 0,C 180,E1 -17749.403,E2 -17749.403} C_VEL
LIN {X 0,Y 276.989,Z 731.432,A -85,B 0,C 180,E1 -17751.196,E2 -17751.196} C_VEL
LIN {X 0,Y 279.108,Z 720.03,A -85,B 0,C 180,E1 -17752.776,E2 -17752.776} C_VEL
LIN {X 0,Y 280.865,Z 708.805,A -85,B 0,C 180,E1 -17753.992,E2 -17753.992} C_VEL
LIN {X 0,Y 282.355,Z 697.264,A -85,B 0,C 180,E1 -17754.934,E2 -17754.934} C_VEL
LIN {X 0,Y 283.644,Z 684.055,A -85,B 0,C 180,E1 -17755.696,E2 -17755.696} C_VEL
LIN {X 0,Y 284.42,Z 671.092,A -85,B 0,C 180,E1 -17756.162,E2 -17756.162} C_VEL
LIN {X 0,Y 286.174,Z 610.237,A -85,B 0,C 180,E1 -17757.67,E2 -17757.67} C_VEL
LIN {X 0,Y 282.431,Z 578.935,A -85,B 0,C 180,E1 -17758.975,E2 -17758.975} C_VEL
LIN {X 0,Y 279.247,Z 559.109,A -85,B 0,C 180,E1 -17759.94,E2 -17759.94} C_VEL
LIN {X 0,Y 278.447,Z 554.771,A -85,B 0,C 180,E1 -17760.497,E2 -17760.497} C_VEL
LIN {X 0,Y 273.09,Z 537.108,A -85,B 0,C 180,E1 -17763.041,E2 -17763.041} C_VEL
LIN {X 0,Y 271.323,Z 531.019,A -85,B 0,C 180,E1 -17764.016,E2 -17764.016} C_VEL
LIN {X 0,Y 270.274,Z 525.809,A -85,B 0,C 180,E1 -17765.692,E2 -17765.692} C_VEL
LIN {X 0,Y 270.195,Z 525.789,A -85,B 0,C 180,E1 -17768.71,E2 -17768.71} C_VEL
LIN {X 0,Y 270.168,Z 525.823,A -85,B 0,C 180,E1 -17773.25,E2 -17773.25} C_VEL
LIN {X 0,Y 270.191,Z 525.819,A -85,B 0,C 180,E1 -17777.446,E2 -17777.446} C_VEL
LIN {X 0,Y 270.241,Z 525.821,A -85,B 0,C 180,E1 -17781.38,E2 -17781.38} C_VEL
LIN {X 0,Y 270.211,Z 525.82,A -85,B 0,C 180,E1 -17785.096,E2 -17785.096} C_VEL
LIN {X 0,Y 270.196,Z 525.807,A -85,B 0,C 180,E1 -17789.13,E2 -17789.13} C_VEL
LIN {X 0,Y 270.26,Z 525.819,A -85,B 0,C 180,E1 -17792.145,E2 -17792.145} C_VEL
LIN {X 0,Y 270.231,Z 525.797,A -85,B 0,C 180,E1 -17795.538,E2 -17795.538} C_VEL
LIN {X 0,Y 270.295,Z 525.814,A -85,B 0,C 180,E1 -17800.244,E2 -17800.244} C_VEL
LIN {X 0,Y 270.39,Z 525.784,A -85,B 0,C 180,E1 -17804.935,E2 -17804.935} C_VEL
LIN {X 0,Y 270.436,Z 525.786,A -85,B 0,C 180,E1 -17809.519,E2 -17809.519} C_VEL
LIN {X 0,Y 270.603,Z 525.749,A -85,B 0,C 180,E1 -17812.539,E2 -17812.539} C_VEL
LIN {X 0,Y 270.782,Z 525.733,A -85,B 0,C 180,E1 -17818.513,E2 -17818.513} C_VEL
LIN {X 0,Y 270.782,Z 525.73,A -85,B 0,C 180,E1 -17821.488,E2 -17821.488} C_VEL
LIN {X 0,Y 270.593,Z 525.751,A -85,B 0,C 180,E1 -17827.462,E2 -17827.462} C_VEL
LIN {X 0,Y 270.407,Z 525.791,A -85,B 0,C 180,E1 -17830.483,E2 -17830.483} C_VEL
LIN {X 0,Y 270.391,Z 525.781,A -85,B 0,C 180,E1 -17835.066,E2 -17835.066} C_VEL
LIN {X 0,Y 270.297,Z 525.816,A -85,B 0,C 180,E1 -17839.756,E2 -17839.756} C_VEL
LIN {X 0,Y 270.27,Z 525.804,A -85,B 0,C 180,E1 -17844.586,E2 -17844.586} C_VEL
LIN {X 0,Y 270.272,Z 525.814,A -85,B 0,C 180,E1 -17847.909,E2 -17847.909} C_VEL
LIN {X 0,Y 270.182,Z 525.825,A -85,B 0,C 180,E1 -17851.349,E2 -17851.349} C_VEL
LIN {X 0,Y 270.199,Z 525.815,A -85,B 0,C 180,E1 -17854.907,E2 -17854.907} C_VEL
LIN {X 0,Y 270.195,Z 525.824,A -85,B 0,C 180,E1 -17858.711,E2 -17858.711} C_VEL
LIN {X 0,Y 270.17,Z 525.827,A -85,B 0,C 180,E1 -17863.252,E2 -17863.252} C_VEL
LIN {X 0,Y 270.174,Z 525.827,A -85,B 0,C 180,E1 -17867.443,E2 -17867.443} C_VEL
LIN {X 0,Y 270.193,Z 525.864,A -85,B 0,C 180,E1 -17870.538,E2 -17870.538} C_VEL
LIN {X 0,Y 273.395,Z 536.392,A -85,B 0,C 180,E1 -17873.755,E2 -17873.755} C_VEL
LIN {X 0,Y 276.525,Z 547.985,A -85,B 0,C 180,E1 -17877.005,E2 -17877.005} C_VEL
LIN {X 0,Y 277.204,Z 550.969,A -85,B 0,C 180,E1 -17877.756,E2 -17877.756} C_VEL
LIN {X 0,Y 283.24,Z 564.909,A -85,B 0,C 180,E1 -17878.896,E2 -17878.896} C_VEL
LIN {X 0,Y 287.46,Z 588.411,A -85,B 0,C 180,E1 -17880.044,E2 -17880.044} C_VEL
LIN {X 0,Y 284.983,Z 661.661,A -85,B 0,C 180,E1 -17881.867,E2 -17881.867} C_VEL
LIN {X 0,Y 284.056,Z 674.973,A -85,B 0,C 180,E1 -17882.461,E2 -17882.461} C_VEL
LIN {X 0,Y 282.835,Z 687.572,A -85,B 0,C 180,E1 -17883.332,E2 -17883.332} C_VEL
LIN {X 0,Y 281.351,Z 699.529,A -85,B 0,C 180,E1 -17884.455,E2 -17884.455} C_VEL
LIN {X 0,Y 279.481,Z 711.148,A -85,B 0,C 180,E1 -17885.882,E2 -17885.882} C_VEL
LIN {X 0,Y 277.502,Z 721.423,A -85,B 0,C 180,E1 -17887.478,E2 -17887.478} C_VEL
LIN {X 0,Y 275.721,Z 729.837,A -85,B 0,C 180,E1 -17889.093,E2 -17889.093} C_VEL
LIN {X 0,Y 273.976,Z 737.582,A -85,B 0,C 180,E1 -17890.91,E2 -17890.91} C_VEL
LIN {X 0,Y 272.35,Z 745.079,A -85,B 0,C 180,E1 -17893.103,E2 -17893.103} C_VEL
LIN {X 0,Y 271.272,Z 750.292,A -85,B 0,C 180,E1 -17894.985,E2 -17894.985} C_VEL
LIN {X 0,Y 270.018,Z 755.266,A -85,B 0,C 180,E1 -17897.219,E2 -17897.219} C_VEL
LIN {X 0,Y 269.241,Z 759.095,A -85,B 0,C 180,E1 -17899.472,E2 -17899.472} C_VEL
LIN {X 0,Y 268.85,Z 761.056,A -85,B 0,C 180,E1 -17900.976,E2 -17900.976} C_VEL
LIN {X 0,Y 268.542,Z 762.608,A -85,B 0,C 180,E1 -17902.481,E2 -17902.481} C_VEL
LIN {X 0,Y 268.27,Z 764.058,A -85,B 0,C 180,E1 -17904.572,E2 -17904.572} C_VEL
LIN {X 0,Y 268.217,Z 764.777,A -85,B 0,C 180,E1 -17906.996,E2 -17906.996} C_VEL
LIN {X 0,Y 268.206,Z 764.721,A -85,B 0,C 180,E1 -17908.498,E2 -17908.498} C_VEL
LIN {X 0,Y 268.207,Z 764.261,A -85,B 0,C 180,E1 -17910,E2 -17910} C_VEL
LIN {X 0,Y 268.482,Z 762.115,A -85,B 0,C 180,E1 -17913.001,E2 -17913.001} C_VEL
LIN {X 0,Y 268.911,Z 759.422,A -85,B 0,C 180,E1 -17915.248,E2 -17915.248} C_VEL
LIN {X 0,Y 269.521,Z 755.269,A -85,B 0,C 180,E1 -17917.737,E2 -17917.737} C_VEL
LIN {X 0,Y 270.277,Z 750.907,A -85,B 0,C 180,E1 -17919.731,E2 -17919.731} C_VEL
LIN {X 0,Y 271.444,Z 744.835,A -85,B 0,C 180,E1 -17921.954,E2 -17921.954} C_VEL
LIN {X 0,Y 272.947,Z 737.223,A -85,B 0,C 180,E1 -17924.159,E2 -17924.159} C_VEL
LIN {X 0,Y 274.764,Z 727.71,A -85,B 0,C 180,E1 -17926.341,E2 -17926.341} C_VEL
LIN {X 0,Y 276.474,Z 717.843,A -85,B 0,C 180,E1 -17928.143,E2 -17928.143} C_VEL
LIN {X 0,Y 278.274,Z 706.725,A -85,B 0,C 180,E1 -17929.742,E2 -17929.742} C_VEL
LIN {X 0,Y 279.701,Z 695.854,A -85,B 0,C 180,E1 -17930.98,E2 -17930.98} C_VEL
LIN {X 0,Y 281.046,Z 684.901,A -85,B 0,C 180,E1 -17931.933,E2 -17931.933} C_VEL
LIN {X 0,Y 282.01,Z 671.981,A -85,B 0,C 180,E1 -17932.766,E2 -17932.766} C_VEL
LIN {X 0,Y 282.722,Z 658.911,A -85,B 0,C 180,E1 -17933.305,E2 -17933.305} C_VEL
LIN {X 0,Y 284.794,Z 586.097,A -85,B 0,C 180,E1 -17935.125,E2 -17935.125} C_VEL
LIN {X 0,Y 280.907,Z 563.113,A -85,B 0,C 180,E1 -17936.165,E2 -17936.165} C_VEL
LIN {X 0,Y 279.877,Z 558.871,A -85,B 0,C 180,E1 -17936.394,E2 -17936.394} C_VEL
LIN {X 0,Y 276.665,Z 550.656,A -85,B 0,C 180,E1 -17937.002,E2 -17937.002} C_VEL
LIN {X 0,Y 274.002,Z 539.145,A -85,B 0,C 180,E1 -17940.009,E2 -17940.009} C_VEL
LIN {X 0,Y 270.613,Z 527.438,A -85,B 0,C 180,E1 -17943.366,E2 -17943.366} C_VEL
LIN {X 0,Y 270.226,Z 525.82,A -85,B 0,C 180,E1 -17943.87,E2 -17943.87} C_VEL
LIN {X 0,Y 270.241,Z 525.815,A -85,B 0,C 180,E1 -17946.736,E2 -17946.736} C_VEL
LIN {X 0,Y 270.249,Z 525.812,A -85,B 0,C 180,E1 -17951.047,E2 -17951.047} C_VEL
LIN {X 0,Y 270.187,Z 525.812,A -85,B 0,C 180,E1 -17955.386,E2 -17955.386} C_VEL
LIN {X 0,Y 270.213,Z 525.826,A -85,B 0,C 180,E1 -17958.019,E2 -17958.019} C_VEL
LIN {X 0,Y 279.766,Z 552.938,A -85,B 0,C 180,E1 -17959.611,E2 -17959.611} C_VEL
LIN {X 0,Y 277.544,Z 613.877,A -85,B 0,C 180,E1 -17961.694,E2 -17961.694} C_VEL
LIN {X 0,Y 276.685,Z 617.761,A -85,B 0,C 180,E1 -17961.796,E2 -17961.796} C_VEL
LIN {X 0,Y 270.528,Z 629.751,A -85,B 0,C 180,E1 -17962.058,E2 -17962.058} C_VEL
LIN {X 0,Y 269.832,Z 633.552,A -85,B 0,C 180,E1 -17962.251,E2 -17962.251} C_VEL
LIN {X 0,Y 269.064,Z 646.496,A -85,B 0,C 180,E1 -17963.176,E2 -17963.176} C_VEL
LIN {X 0,Y 267.934,Z 660.254,A -85,B 0,C 180,E1 -17964.507,E2 -17964.507} C_VEL
LIN {X 0,Y 266.808,Z 671.802,A -85,B 0,C 180,E1 -17965.961,E2 -17965.961} C_VEL
LIN {X 0,Y 265.718,Z 682.599,A -85,B 0,C 180,E1 -17967.655,E2 -17967.655} C_VEL
LIN {X 0,Y 264.737,Z 691.065,A -85,B 0,C 180,E1 -17969.267,E2 -17969.267} C_VEL
LIN {X 0,Y 263.762,Z 700.044,A -85,B 0,C 180,E1 -17971.339,E2 -17971.339} C_VEL
LIN {X 0,Y 262.84,Z 708.599,A -85,B 0,C 180,E1 -17973.82,E2 -17973.82} C_VEL
LIN {X 0,Y 262.215,Z 715.366,A -85,B 0,C 180,E1 -17976.294,E2 -17976.294} C_VEL
LIN {X 0,Y 261.739,Z 720.545,A -85,B 0,C 180,E1 -17978.746,E2 -17978.746} C_VEL
LIN {X 0,Y 261.5,Z 724.422,A -85,B 0,C 180,E1 -17981.185,E2 -17981.185} C_VEL
LIN {X 0,Y 261.454,Z 726.365,A -85,B 0,C 180,E1 -17982.801,E2 -17982.801} C_VEL
LIN {X 0,Y 261.636,Z 728.371,A -85,B 0,C 180,E1 -17985.24,E2 -17985.24} C_VEL
LIN {X 0,Y 261.98,Z 729.298,A -85,B 0,C 180,E1 -17987.607,E2 -17987.607} C_VEL
LIN {X 0,Y 262.394,Z 729.374,A -85,B 0,C 180,E1 -17989.193,E2 -17989.193} C_VEL
LIN {X 0,Y 263.121,Z 728.796,A -85,B 0,C 180,E1 -17991.208,E2 -17991.208} C_VEL
LIN {X 0,Y 264.337,Z 726.93,A -85,B 0,C 180,E1 -17993.895,E2 -17993.895} C_VEL
LIN {X 0,Y 265.74,Z 724.19,A -85,B 0,C 180,E1 -17996.209,E2 -17996.209} C_VEL
LIN {X 0,Y 267.455,Z 720.37,A -85,B 0,C 180,E1 -17998.494,E2 -17998.494} C_VEL
LIN {X 0,Y 269.5,Z 715.41,A -85,B 0,C 180,E1 -18000.747,E2 -18000.747} C_VEL
LIN {X 0,Y 271.841,Z 709.139,A -85,B 0,C 180,E1 -18002.964,E2 -18002.964} C_VEL
LIN {X 0,Y 274.606,Z 701.269,A -85,B 0,C 180,E1 -18005.14,E2 -18005.14} C_VEL
LIN {X 0,Y 277.623,Z 691.539,A -85,B 0,C 180,E1 -18007.271,E2 -18007.271} C_VEL
LIN {X 0,Y 280.511,Z 681.433,A -85,B 0,C 180,E1 -18009.009,E2 -18009.009} C_VEL
LIN {X 0,Y 282.885,Z 671.622,A -85,B 0,C 180,E1 -18010.376,E2 -18010.376} C_VEL
LIN {X 0,Y 285.416,Z 659.277,A -85,B 0,C 180,E1 -18011.721,E2 -18011.721} C_VEL
LIN {X 0,Y 287.458,Z 646.526,A -85,B 0,C 180,E1 -18012.81,E2 -18012.81} C_VEL
LIN {X 0,Y 289.029,Z 633.028,A -85,B 0,C 180,E1 -18013.649,E2 -18013.649} C_VEL
LIN {X 0,Y 291.778,Z 602.617,A -85,B 0,C 180,E1 -18014.848,E2 -18014.848} C_VEL
LIN {X 0,Y 294.54,Z 573.424,A -85,B 0,C 180,E1 -18015.951,E2 -18015.951} C_VEL
LIN {X 0,Y 289.996,Z 564.913,A -85,B 0,C 180,E1 -18017.652,E2 -18017.652} C_VEL
LIN {X 0,Y 285.89,Z 558.307,A -85,B 0,C 180,E1 -18019.327,E2 -18019.327} C_VEL
LIN {X 0,Y 281.355,Z 551.829,A -85,B 0,C 180,E1 -18021.394,E2 -18021.394} C_VEL
LIN {X 0,Y 278.048,Z 547.669,A -85,B 0,C 180,E1 -18023.107,E2 -18023.107} C_VEL
LIN {X 0,Y 274.952,Z 543.914,A -85,B 0,C 180,E1 -18024.978,E2 -18024.978} C_VEL
LIN {X 0,Y 271.303,Z 540.276,A -85,B 0,C 180,E1 -18027.688,E2 -18027.688} C_VEL
LIN {X 0,Y 270.463,Z 539.322,A -85,B 0,C 180,E1 -18028.466,E2 -18028.466} C_VEL
LIN {X 0,Y 267.153,Z 536.921,A -85,B 0,C 180,E1 -18032.669,E2 -18032.669} C_VEL
LIN {X 0,Y 266.556,Z 536.35,A -85,B 0,C 180,E1 -18034.55,E2 -18034.55} C_VEL
LIN {X 0,Y 266.958,Z 537.605,A -85,B 0,C 180,E1 -18037.836,E2 -18037.836} C_VEL
LIN {X 0,Y 267.908,Z 540.38,A -85,B 0,C 180,E1 -18041.868,E2 -18041.868} C_VEL
LIN {X 0,Y 270.895,Z 545.999,A -85,B 0,C 180,E1 -18045.416,E2 -18045.416} C_VEL
LIN {X 0,Y 274.052,Z 550.65,A -85,B 0,C 180,E1 -18047.842,E2 -18047.842} C_VEL
LIN {X 0,Y 277.882,Z 557.344,A -85,B 0,C 180,E1 -18050.272,E2 -18050.272} C_VEL
LIN {X 0,Y 281.992,Z 565.131,A -85,B 0,C 180,E1 -18052.459,E2 -18052.459} C_VEL
LIN {X 0,Y 285.039,Z 571.54,A -85,B 0,C 180,E1 -18053.905,E2 -18053.905} C_VEL
LIN {X 0,Y 287.986,Z 578.233,A -85,B 0,C 180,E1 -18055.22,E2 -18055.22} C_VEL
LIN {X 0,Y 289.29,Z 582.138,A -85,B 0,C 180,E1 -18055.811,E2 -18055.811} C_VEL
LIN {X 0,Y 290.815,Z 596.423,A -85,B 0,C 180,E1 -18057.095,E2 -18057.095} C_VEL
LIN {X 0,Y 291.568,Z 608.511,A -85,B 0,C 180,E1 -18057.976,E2 -18057.976} C_VEL
LIN {X 0,Y 291.621,Z 614.972,A -85,B 0,C 180,E1 -18058.358,E2 -18058.358} C_VEL
LIN {X 0,Y 287.36,Z 661.215,A -85,B 0,C 180,E1 -18060.112,E2 -18060.112} C_VEL
LIN {X 0,Y 285.208,Z 675.547,A -85,B 0,C 180,E1 -18060.879,E2 -18060.879} C_VEL
LIN {X 0,Y 282.396,Z 689.938,A -85,B 0,C 180,E1 -18061.983,E2 -18061.983} C_VEL
LIN {X 0,Y 279.374,Z 702.578,A -85,B 0,C 180,E1 -18063.278,E2 -18063.278} C_VEL
LIN {X 0,Y 276.29,Z 713.975,A -85,B 0,C 180,E1 -18064.782,E2 -18064.782} C_VEL
LIN {X 0,Y 273.299,Z 724.393,A -85,B 0,C 180,E1 -18066.511,E2 -18066.511} C_VEL
LIN {X 0,Y 270.086,Z 734.611,A -85,B 0,C 180,E1 -18068.636,E2 -18068.636} C_VEL
LIN {X 0,Y 267.487,Z 742.96,A -85,B 0,C 180,E1 -18070.828,E2 -18070.828} C_VEL
LIN {X 0,Y 265.103,Z 750.92,A -85,B 0,C 180,E1 -18073.442,E2 -18073.442} C_VEL
LIN {X 0,Y 263.635,Z 758.714,A -85,B 0,C 180,E1 -18075.725,E2 -18075.725} C_VEL
LIN {X 0,Y 262.337,Z 765.827,A -85,B 0,C 180,E1 -18078.409,E2 -18078.409} C_VEL
LIN {X 0,Y 261.674,Z 770.555,A -85,B 0,C 180,E1 -18080.727,E2 -18080.727} C_VEL
LIN {X 0,Y 261.311,Z 774.152,A -85,B 0,C 180,E1 -18083.049,E2 -18083.049} C_VEL
LIN {X 0,Y 261.105,Z 776.72,A -85,B 0,C 180,E1 -18085.368,E2 -18085.368} C_VEL
LIN {X 0,Y 261.129,Z 777.919,A -85,B 0,C 180,E1 -18086.914,E2 -18086.914} C_VEL
LIN {X 0,Y 261.144,Z 778.665,A -85,B 0,C 180,E1 -18088.458,E2 -18088.458} C_VEL
LIN {X 0,Y 261.135,Z 779.011,A -85,B 0,C 180,E1 -18090,E2 -18090} C_VEL
LIN {X 0,Y 261.137,Z 778.968,A -85,B 0,C 180,E1 -18091.542,E2 -18091.542} C_VEL
LIN {X 0,Y 261.129,Z 778.521,A -85,B 0,C 180,E1 -18093.086,E2 -18093.086} C_VEL
LIN {X 0,Y 261.221,Z 776.346,A -85,B 0,C 180,E1 -18096.178,E2 -18096.178} C_VEL
LIN {X 0,Y 261.548,Z 773.617,A -85,B 0,C 180,E1 -18098.499,E2 -18098.499} C_VEL
LIN {X 0,Y 262.159,Z 769.862,A -85,B 0,C 180,E1 -18100.816,E2 -18100.816} C_VEL
LIN {X 0,Y 263.083,Z 764.971,A -85,B 0,C 180,E1 -18103.124,E2 -18103.124} C_VEL
LIN {X 0,Y 264.543,Z 758.803,A -85,B 0,C 180,E1 -18105.406,E2 -18105.406} C_VEL
LIN {X 0,Y 266.287,Z 751.093,A -85,B 0,C 180,E1 -18107.668,E2 -18107.668} C_VEL
LIN {X 0,Y 267.927,Z 743.203,A -85,B 0,C 180,E1 -18109.538,E2 -18109.538} C_VEL
LIN {X 0,Y 269.926,Z 733.562,A -85,B 0,C 180,E1 -18111.377,E2 -18111.377} C_VEL
LIN {X 0,Y 272.119,Z 722.835,A -85,B 0,C 180,E1 -18112.993,E2 -18112.993} C_VEL
LIN {X 0,Y 273.863,Z 712.333,A -85,B 0,C 180,E1 -18114.242,E2 -18114.242} C_VEL
LIN {X 0,Y 275.691,Z 699.716,A -85,B 0,C 180,E1 -18115.377,E2 -18115.377} C_VEL
LIN {X 0,Y 277.082,Z 687.011,A -85,B 0,C 180,E1 -18116.199,E2 -18116.199} C_VEL
LIN {X 0,Y 278.009,Z 674.612,A -85,B 0,C 180,E1 -18116.711,E2 -18116.711} C_VEL
LIN {X 0,Y 279.964,Z 611.141,A -85,B 0,C 180,E1 -18118.336,E2 -18118.336} C_VEL
LIN {X 0,Y 276.15,Z 579.176,A -85,B 0,C 180,E1 -18119.717,E2 -18119.717} C_VEL
LIN {X 0,Y 273.002,Z 559.943,A -85,B 0,C 180,E1 -18120.686,E2 -18120.686} C_VEL
LIN {X 0,Y 272.007,Z 556.638,A -85,B 0,C 180,E1 -18121.114,E2 -18121.114} C_VEL
LIN {X 0,Y 267.437,Z 540.834,A -85,B 0,C 180,E1 -18123.494,E2 -18123.494} C_VEL
LIN {X 0,Y 263.412,Z 527.515,A -85,B 0,C 180,E1 -18125.68,E2 -18125.68} C_VEL
LIN {X 0,Y 263.218,Z 526.68,A -85,B 0,C 180,E1 -18125.972,E2 -18125.972} C_VEL
LIN {X 0,Y 263.103,Z 526.684,A -85,B 0,C 180,E1 -18129.872,E2 -18129.872} C_VEL
LIN {X 0,Y 263.126,Z 526.699,A -85,B 0,C 180,E1 -18133.982,E2 -18133.982} C_VEL
LIN {X 0,Y 263.152,Z 526.692,A -85,B 0,C 180,E1 -18138.398,E2 -18138.398} C_VEL
LIN {X 0,Y 263.185,Z 526.693,A -85,B 0,C 180,E1 -18142.107,E2 -18142.107} C_VEL
LIN {X 0,Y 263.18,Z 526.702,A -85,B 0,C 180,E1 -18145.89,E2 -18145.89} C_VEL
LIN {X 0,Y 263.146,Z 526.685,A -85,B 0,C 180,E1 -18149.506,E2 -18149.506} C_VEL
LIN {X 0,Y 263.187,Z 526.7,A -85,B 0,C 180,E1 -18153.002,E2 -18153.002} C_VEL
LIN {X 0,Y 263.148,Z 526.678,A -85,B 0,C 180,E1 -18156.384,E2 -18156.384} C_VEL
LIN {X 0,Y 263.257,Z 526.691,A -85,B 0,C 180,E1 -18159.693,E2 -18159.693} C_VEL
LIN {X 0,Y 263.339,Z 526.657,A -85,B 0,C 180,E1 -18164.522,E2 -18164.522} C_VEL
LIN {X 0,Y 263.368,Z 526.668,A -85,B 0,C 180,E1 -18169.234,E2 -18169.234} C_VEL
LIN {X 0,Y 263.564,Z 526.623,A -85,B 0,C 180,E1 -18172.338,E2 -18172.338} C_VEL
LIN {X 0,Y 263.746,Z 526.609,A -85,B 0,C 180,E1 -18178.473,E2 -18178.473} C_VEL
LIN {X 0,Y 263.747,Z 526.607,A -85,B 0,C 180,E1 -18181.527,E2 -18181.527} C_VEL
LIN {X 0,Y 263.553,Z 526.626,A -85,B 0,C 180,E1 -18187.663,E2 -18187.663} C_VEL
LIN {X 0,Y 263.349,Z 526.672,A -85,B 0,C 180,E1 -18190.767,E2 -18190.767} C_VEL
LIN {X 0,Y 263.339,Z 526.656,A -85,B 0,C 180,E1 -18195.479,E2 -18195.479} C_VEL
LIN {X 0,Y 263.259,Z 526.692,A -85,B 0,C 180,E1 -18200.307,E2 -18200.307} C_VEL
LIN {X 0,Y 263.206,Z 526.691,A -85,B 0,C 180,E1 -18205.292,E2 -18205.292} C_VEL
LIN {X 0,Y 263.181,Z 526.686,A -85,B 0,C 180,E1 -18208.73,E2 -18208.73} C_VEL
LIN {X 0,Y 263.131,Z 526.709,A -85,B 0,C 180,E1 -18212.289,E2 -18212.289} C_VEL
LIN {X 0,Y 263.18,Z 526.703,A -85,B 0,C 180,E1 -18216.764,E2 -18216.764} C_VEL
LIN {X 0,Y 263.124,Z 526.716,A -85,B 0,C 180,E1 -18221.595,E2 -18221.595} C_VEL
LIN {X 0,Y 263.127,Z 526.708,A -85,B 0,C 180,E1 -18226.018,E2 -18226.018} C_VEL
LIN {X 0,Y 263.155,Z 526.901,A -85,B 0,C 180,E1 -18229.654,E2 -18229.654} C_VEL
LIN {X 0,Y 266.468,Z 537.274,A -85,B 0,C 180,E1 -18232.923,E2 -18232.923} C_VEL
LIN {X 0,Y 269.292,Z 547.679,A -85,B 0,C 180,E1 -18235.946,E2 -18235.946} C_VEL
LIN {X 0,Y 270.23,Z 551.244,A -85,B 0,C 180,E1 -18236.863,E2 -18236.863} C_VEL
LIN {X 0,Y 277.338,Z 567.426,A -85,B 0,C 180,E1 -18238.261,E2 -18238.261} C_VEL
LIN {X 0,Y 281.171,Z 588.635,A -85,B 0,C 180,E1 -18239.339,E2 -18239.339} C_VEL
LIN {X 0,Y 278.655,Z 662.452,A -85,B 0,C 180,E1 -18241.227,E2 -18241.227} C_VEL
LIN {X 0,Y 277.71,Z 675.408,A -85,B 0,C 180,E1 -18241.828,E2 -18241.828} C_VEL
LIN {X 0,Y 276.498,Z 687.412,A -85,B 0,C 180,E1 -18242.671,E2 -18242.671} C_VEL
LIN {X 0,Y 274.892,Z 699.814,A -85,B 0,C 180,E1 -18243.854,E2 -18243.854} C_VEL
LIN {X 0,Y 273,Z 711.139,A -85,B 0,C 180,E1 -18245.271,E2 -18245.271} C_VEL
LIN {X 0,Y 270.943,Z 721.448,A -85,B 0,C 180,E1 -18246.901,E2 -18246.901} C_VEL
LIN {X 0,Y 269.076,Z 729.89,A -85,B 0,C 180,E1 -18248.552,E2 -18248.552} C_VEL
LIN {X 0,Y 267.247,Z 737.659,A -85,B 0,C 180,E1 -18250.41,E2 -18250.41} C_VEL
LIN {X 0,Y 265.724,Z 744.438,A -85,B 0,C 180,E1 -18252.408,E2 -18252.408} C_VEL
LIN {X 0,Y 264.399,Z 750.411,A -85,B 0,C 180,E1 -18254.585,E2 -18254.585} C_VEL
LIN {X 0,Y 263.066,Z 755.403,A -85,B 0,C 180,E1 -18256.875,E2 -18256.875} C_VEL
LIN {X 0,Y 262.245,Z 759.246,A -85,B 0,C 180,E1 -18259.188,E2 -18259.188} C_VEL
LIN {X 0,Y 261.826,Z 761.213,A -85,B 0,C 180,E1 -18260.732,E2 -18260.732} C_VEL
LIN {X 0,Y 261.501,Z 762.772,A -85,B 0,C 180,E1 -18262.278,E2 -18262.278} C_VEL
LIN {X 0,Y 261.175,Z 764.35,A -85,B 0,C 180,E1 -18264.655,E2 -18264.655} C_VEL
LIN {X 0,Y 261.131,Z 764.965,A -85,B 0,C 180,E1 -18266.915,E2 -18266.915} C_VEL
LIN {X 0,Y 261.133,Z 764.914,A -85,B 0,C 180,E1 -18268.458,E2 -18268.458} C_VEL
LIN {X 0,Y 261.133,Z 764.466,A -85,B 0,C 180,E1 -18270,E2 -18270} C_VEL
LIN {X 0,Y 261.42,Z 762.332,A -85,B 0,C 180,E1 -18273.082,E2 -18273.082} C_VEL
LIN {X 0,Y 261.854,Z 759.652,A -85,B 0,C 180,E1 -18275.39,E2 -18275.39} C_VEL
LIN {X 0,Y 262.403,Z 755.965,A -85,B 0,C 180,E1 -18277.696,E2 -18277.696} C_VEL
LIN {X 0,Y 263.287,Z 751.163,A -85,B 0,C 180,E1 -18279.992,E2 -18279.992} C_VEL
LIN {X 0,Y 264.501,Z 745.106,A -85,B 0,C 180,E1 -18282.272,E2 -18282.272} C_VEL
LIN {X 0,Y 266.071,Z 737.52,A -85,B 0,C 180,E1 -18284.532,E2 -18284.532} C_VEL
LIN {X 0,Y 267.984,Z 728.025,A -85,B 0,C 180,E1 -18286.767,E2 -18286.767} C_VEL
LIN {X 0,Y 269.77,Z 718.195,A -85,B 0,C 180,E1 -18288.61,E2 -18288.61} C_VEL
LIN {X 0,Y 271.634,Z 707.108,A -85,B 0,C 180,E1 -18290.245,E2 -18290.245} C_VEL
LIN {X 0,Y 273.11,Z 696.281,A -85,B 0,C 180,E1 -18291.512,E2 -18291.512} C_VEL
LIN {X 0,Y 274.502,Z 685.402,A -85,B 0,C 180,E1 -18292.484,E2 -18292.484} C_VEL
LIN {X 0,Y 275.472,Z 672.915,A -85,B 0,C 180,E1 -18293.322,E2 -18293.322} C_VEL
LIN {X 0,Y 276.25,Z 659.613,A -85,B 0,C 180,E1 -18293.892,E2 -18293.892} C_VEL
LIN {X 0,Y 278.437,Z 587.146,A -85,B 0,C 180,E1 -18295.742,E2 -18295.742} C_VEL
LIN {X 0,Y 274.767,Z 565.121,A -85,B 0,C 180,E1 -18296.769,E2 -18296.769} C_VEL
LIN {X 0,Y 273.637,Z 560.858,A -85,B 0,C 180,E1 -18297.019,E2 -18297.019} C_VEL
LIN {X 0,Y 269.609,Z 550.751,A -85,B 0,C 180,E1 -18297.809,E2 -18297.809} C_VEL
LIN {X 0,Y 266.805,Z 539.296,A -85,B 0,C 180,E1 -18300.906,E2 -18300.906} C_VEL
LIN {X 0,Y 263.184,Z 526.701,A -85,B 0,C 180,E1 -18304.658,E2 -18304.658} C_VEL
LIN {X 0,Y 263.188,Z 526.7,A -85,B 0,C 180,E1 -18307.891,E2 -18307.891} C_VEL
LIN {X 0,Y 263.167,Z 526.702,A -85,B 0,C 180,E1 -18311.884,E2 -18311.884} C_VEL
LIN {X 0,Y 263.137,Z 526.694,A -85,B 0,C 180,E1 -18316.146,E2 -18316.146} C_VEL
LIN {X 0,Y 263.168,Z 526.704,A -85,B 0,C 180,E1 -18317.577,E2 -18317.577} C_VEL
LIN {X 0,Y 272.931,Z 554.509,A -85,B 0,C 180,E1 -18319.28,E2 -18319.28} C_VEL
LIN {X 0,Y 270.257,Z 624.938,A -85,B 0,C 180,E1 -18321.798,E2 -18321.798} C_VEL
LIN {X 0,Y 269.832,Z 633.552,A -85,B 0,C 180,E1 -18322.251,E2 -18322.251} C_VEL
LIN {X 0,Y 269.058,Z 639.192,A -85,B 0,C 180,E1 -18322.582,E2 -18322.582} C_VEL
LIN {X 0,Y 265.62,Z 648.139,A -85,B 0,C 180,E1 -18323.139,E2 -18323.139} C_VEL
LIN {X 0,Y 261.934,Z 656.805,A -85,B 0,C 180,E1 -18323.853,E2 -18323.853} C_VEL
LIN {X 0,Y 260.794,Z 662.011,A -85,B 0,C 180,E1 -18324.424,E2 -18324.424} C_VEL
LIN {X 0,Y 259.553,Z 674.181,A -85,B 0,C 180,E1 -18326.049,E2 -18326.049} C_VEL
LIN {X 0,Y 258.58,Z 683.94,A -85,B 0,C 180,E1 -18327.664,E2 -18327.664} C_VEL
LIN {X 0,Y 257.401,Z 693.785,A -85,B 0,C 180,E1 -18329.66,E2 -18329.66} C_VEL
LIN {X 0,Y 256.48,Z 701.952,A -85,B 0,C 180,E1 -18331.685,E2 -18331.685} C_VEL
LIN {X 0,Y 255.694,Z 709.316,A -85,B 0,C 180,E1 -18333.91,E2 -18333.91} C_VEL
LIN {X 0,Y 255.17,Z 715.035,A -85,B 0,C 180,E1 -18336.03,E2 -18336.03} C_VEL
LIN {X 0,Y 254.74,Z 719.647,A -85,B 0,C 180,E1 -18338.133,E2 -18338.133} C_VEL
LIN {X 0,Y 254.446,Z 723.946,A -85,B 0,C 180,E1 -18340.643,E2 -18340.643} C_VEL
LIN {X 0,Y 254.355,Z 726.135,A -85,B 0,C 180,E1 -18342.305,E2 -18342.305} C_VEL
LIN {X 0,Y 254.53,Z 728.662,A -85,B 0,C 180,E1 -18345.102,E2 -18345.102} C_VEL
LIN {X 0,Y 254.827,Z 729.74,A -85,B 0,C 180,E1 -18347.253,E2 -18347.253} C_VEL
LIN {X 0,Y 255.223,Z 730.011,A -85,B 0,C 180,E1 -18348.886,E2 -18348.886} C_VEL
LIN {X 0,Y 256.038,Z 729.665,A -85,B 0,C 180,E1 -18351.167,E2 -18351.167} C_VEL
LIN {X 0,Y 257.166,Z 728.222,A -85,B 0,C 180,E1 -18353.724,E2 -18353.724} C_VEL
LIN {X 0,Y 258.09,Z 726.747,A -85,B 0,C 180,E1 -18355.314,E2 -18355.314} C_VEL
LIN {X 0,Y 259.165,Z 724.841,A -85,B 0,C 180,E1 -18356.891,E2 -18356.891} C_VEL
LIN {X 0,Y 261.024,Z 721.054,A -85,B 0,C 180,E1 -18359.228,E2 -18359.228} C_VEL
LIN {X 0,Y 263.239,Z 716.08,A -85,B 0,C 180,E1 -18361.53,E2 -18361.53} C_VEL
LIN {X 0,Y 265.762,Z 709.807,A -85,B 0,C 180,E1 -18363.79,E2 -18363.79} C_VEL
LIN {X 0,Y 268.728,Z 702.021,A -85,B 0,C 180,E1 -18366.004,E2 -18366.004} C_VEL
LIN {X 0,Y 271.386,Z 694.118,A -85,B 0,C 180,E1 -18367.814,E2 -18367.814} C_VEL
LIN {X 0,Y 274.385,Z 684.383,A -85,B 0,C 180,E1 -18369.583,E2 -18369.583} C_VEL
LIN {X 0,Y 277.198,Z 673.794,A -85,B 0,C 180,E1 -18371.146,E2 -18371.146} C_VEL
LIN {X 0,Y 279.887,Z 662.065,A -85,B 0,C 180,E1 -18372.508,E2 -18372.508} C_VEL
LIN {X 0,Y 282.163,Z 649.3,A -85,B 0,C 180,E1 -18373.653,E2 -18373.653} C_VEL
LIN {X 0,Y 283.902,Z 636.275,A -85,B 0,C 180,E1 -18374.518,E2 -18374.518} C_VEL
LIN {X 0,Y 285.973,Z 614.284,A -85,B 0,C 180,E1 -18375.478,E2 -18375.478} C_VEL
LIN {X 0,Y 289.84,Z 576.724,A -85,B 0,C 180,E1 -18376.916,E2 -18376.916} C_VEL
LIN {X 0,Y 285.808,Z 568.978,A -85,B 0,C 180,E1 -18378.562,E2 -18378.562} C_VEL
LIN {X 0,Y 281.776,Z 562.613,A -85,B 0,C 180,E1 -18380.323,E2 -18380.323} C_VEL
LIN {X 0,Y 277.984,Z 557.222,A -85,B 0,C 180,E1 -18382.19,E2 -18382.19} C_VEL
LIN {X 0,Y 275.417,Z 553.847,A -85,B 0,C 180,E1 -18383.651,E2 -18383.651} C_VEL
LIN {X 0,Y 272.337,Z 550.053,A -85,B 0,C 180,E1 -18385.657,E2 -18385.657} C_VEL
LIN {X 0,Y 269.26,Z 546.747,A -85,B 0,C 180,E1 -18388.142,E2 -18388.142} C_VEL
LIN {X 0,Y 268.081,Z 545.79,A -85,B 0,C 180,E1 -18389.255,E2 -18389.255} C_VEL
LIN {X 0,Y 265.567,Z 543.754,A -85,B 0,C 180,E1 -18392.947,E2 -18392.947} C_VEL
LIN {X 0,Y 264.99,Z 543.312,A -85,B 0,C 180,E1 -18394.699,E2 -18394.699} C_VEL
LIN {X 0,Y 264.839,Z 544.674,A -85,B 0,C 180,E1 -18398.338,E2 -18398.338} C_VEL
LIN {X 0,Y 266.205,Z 547.181,A -85,B 0,C 180,E1 -18401.611,E2 -18401.611} C_VEL
LIN {X 0,Y 269.043,Z 552.761,A -85,B 0,C 180,E1 -18405.148,E2 -18405.148} C_VEL
LIN {X 0,Y 271.657,Z 556.851,A -85,B 0,C 180,E1 -18407.298,E2 -18407.298} C_VEL
LIN {X 0,Y 275.175,Z 563.299,A -85,B 0,C 180,E1 -18409.7,E2 -18409.7} C_VEL
LIN {X 0,Y 278.951,Z 570.931,A -85,B 0,C 180,E1 -18411.872,E2 -18411.872} C_VEL
LIN {X 0,Y 281.696,Z 577.058,A -85,B 0,C 180,E1 -18413.296,E2 -18413.296} C_VEL
LIN {X 0,Y 284.682,Z 584.228,A -85,B 0,C 180,E1 -18414.715,E2 -18414.715} C_VEL
LIN {X 0,Y 285.169,Z 587.048,A -85,B 0,C 180,E1 -18415.055,E2 -18415.055} C_VEL
LIN {X 0,Y 286.468,Z 601.272,A -85,B 0,C 180,E1 -18416.327,E2 -18416.327} C_VEL
LIN {X 0,Y 286.884,Z 614.396,A -85,B 0,C 180,E1 -18417.263,E2 -18417.263} C_VEL
LIN {X 0,Y 282.448,Z 660.694,A -85,B 0,C 180,E1 -18419.072,E2 -18419.072} C_VEL
LIN {X 0,Y 280.313,Z 674.168,A -85,B 0,C 180,E1 -18419.802,E2 -18419.802} C_VEL
LIN {X 0,Y 277.529,Z 687.639,A -85,B 0,C 180,E1 -18420.826,E2 -18420.826} C_VEL
LIN {X 0,Y 274.312,Z 700.564,A -85,B 0,C 180,E1 -18422.124,E2 -18422.124} C_VEL
LIN {X 0,Y 270.995,Z 712.203,A -85,B 0,C 180,E1 -18423.634,E2 -18423.634} C_VEL
LIN {X 0,Y 268.098,Z 721.789,A -85,B 0,C 180,E1 -18425.202,E2 -18425.202} C_VEL
LIN {X 0,Y 265.141,Z 730.718,A -85,B 0,C 180,E1 -18426.986,E2 -18426.986} C_VEL
LIN {X 0,Y 262.124,Z 739.602,A -85,B 0,C 180,E1 -18429.191,E2 -18429.191} C_VEL
LIN {X 0,Y 259.634,Z 747.088,A -85,B 0,C 180,E1 -18431.533,E2 -18431.533} C_VEL
LIN {X 0,Y 257.97,Z 752.077,A -85,B 0,C 180,E1 -18433.378,E2 -18433.378} C_VEL
LIN {X 0,Y 256.482,Z 759.571,A -85,B 0,C 180,E1 -18435.723,E2 -18435.723} C_VEL
LIN {X 0,Y 255.328,Z 765.58,A -85,B 0,C 180,E1 -18438.086,E2 -18438.086} C_VEL
LIN {X 0,Y 254.625,Z 770.32,A -85,B 0,C 180,E1 -18440.468,E2 -18440.468} C_VEL
LIN {X 0,Y 254.241,Z 773.928,A -85,B 0,C 180,E1 -18442.854,E2 -18442.854} C_VEL
LIN {X 0,Y 254.013,Z 776.506,A -85,B 0,C 180,E1 -18445.239,E2 -18445.239} C_VEL
LIN {X 0,Y 254.024,Z 777.712,A -85,B 0,C 180,E1 -18446.828,E2 -18446.828} C_VEL
LIN {X 0,Y 254.05,Z 778.466,A -85,B 0,C 180,E1 -18448.415,E2 -18448.415} C_VEL
LIN {X 0,Y 254.062,Z 778.818,A -85,B 0,C 180,E1 -18450,E2 -18450} C_VEL
LIN {X 0,Y 254.044,Z 778.779,A -85,B 0,C 180,E1 -18451.585,E2 -18451.585} C_VEL
LIN {X 0,Y 254.023,Z 778.34,A -85,B 0,C 180,E1 -18453.172,E2 -18453.172} C_VEL
LIN {X 0,Y 254.152,Z 776.177,A -85,B 0,C 180,E1 -18456.35,E2 -18456.35} C_VEL
LIN {X 0,Y 254.499,Z 773.459,A -85,B 0,C 180,E1 -18458.736,E2 -18458.736} C_VEL
LIN {X 0,Y 255.145,Z 769.715,A -85,B 0,C 180,E1 -18461.117,E2 -18461.117} C_VEL
LIN {X 0,Y 256.158,Z 764.837,A -85,B 0,C 180,E1 -18463.486,E2 -18463.486} C_VEL
LIN {X 0,Y 257.68,Z 758.684,A -85,B 0,C 180,E1 -18465.827,E2 -18465.827} C_VEL
LIN {X 0,Y 259.5,Z 751.079,A -85,B 0,C 180,E1 -18468.124,E2 -18468.124} C_VEL
LIN {X 0,Y 261.23,Z 743.128,A -85,B 0,C 180,E1 -18470.06,E2 -18470.06} C_VEL
LIN {X 0,Y 263.31,Z 733.512,A -85,B 0,C 180,E1 -18471.942,E2 -18471.942} C_VEL
LIN {X 0,Y 265.592,Z 722.824,A -85,B 0,C 180,E1 -18473.592,E2 -18473.592} C_VEL
LIN {X 0,Y 267.42,Z 712.378,A -85,B 0,C 180,E1 -18474.865,E2 -18474.865} C_VEL
LIN {X 0,Y 269.307,Z 699.83,A -85,B 0,C 180,E1 -18476.023,E2 -18476.023} C_VEL
LIN {X 0,Y 270.748,Z 687.284,A -85,B 0,C 180,E1 -18476.86,E2 -18476.86} C_VEL
LIN {X 0,Y 271.755,Z 673.801,A -85,B 0,C 180,E1 -18477.429,E2 -18477.429} C_VEL
LIN {X 0,Y 273.694,Z 611.237,A -85,B 0,C 180,E1 -18479.068,E2 -18479.068} C_VEL
LIN {X 0,Y 270.092,Z 580.643,A -85,B 0,C 180,E1 -18480.434,E2 -18480.434} C_VEL
LIN {X 0,Y 267.082,Z 562.122,A -85,B 0,C 180,E1 -18481.4,E2 -18481.4} C_VEL
LIN {X 0,Y 265.78,Z 558.917,A -85,B 0,C 180,E1 -18481.684,E2 -18481.684} C_VEL
LIN {X 0,Y 261.279,Z 543.026,A -85,B 0,C 180,E1 -18484.195,E2 -18484.195} C_VEL
LIN {X 0,Y 257.975,Z 531.867,A -85,B 0,C 180,E1 -18486.062,E2 -18486.062} C_VEL
LIN {X 0,Y 256.191,Z 527.851,A -85,B 0,C 180,E1 -18486.879,E2 -18486.879} C_VEL
LIN {X 0,Y 256.153,Z 527.542,A -85,B 0,C 180,E1 -18486.949,E2 -18486.949} C_VEL
LIN {X 0,Y 256.053,Z 527.589,A -85,B 0,C 180,E1 -18491.203,E2 -18491.203} C_VEL
LIN {X 0,Y 256.063,Z 527.591,A -85,B 0,C 180,E1 -18495.528,E2 -18495.528} C_VEL
LIN {X 0,Y 256.082,Z 527.573,A -85,B 0,C 180,E1 -18498.802,E2 -18498.802} C_VEL
LIN {X 0,Y 256.151,Z 527.562,A -85,B 0,C 180,E1 -18502.871,E2 -18502.871} C_VEL
LIN {X 0,Y 256.081,Z 527.587,A -85,B 0,C 180,E1 -18506.709,E2 -18506.709} C_VEL
LIN {X 0,Y 256.134,Z 527.574,A -85,B 0,C 180,E1 -18511.404,E2 -18511.404} C_VEL
LIN {X 0,Y 256.137,Z 527.551,A -85,B 0,C 180,E1 -18515.696,E2 -18515.696} C_VEL
LIN {X 0,Y 256.157,Z 527.575,A -85,B 0,C 180,E1 -18519.104,E2 -18519.104} C_VEL
LIN {X 0,Y 256.255,Z 527.534,A -85,B 0,C 180,E1 -18523.715,E2 -18523.715} C_VEL
LIN {X 0,Y 256.289,Z 527.562,A -85,B 0,C 180,E1 -18527.328,E2 -18527.328} C_VEL
LIN {X 0,Y 256.475,Z 527.51,A -85,B 0,C 180,E1 -18530.56,E2 -18530.56} C_VEL
LIN {X 0,Y 256.481,Z 527.52,A -85,B 0,C 180,E1 -18533.708,E2 -18533.708} C_VEL
LIN {X 0,Y 256.709,Z 527.485,A -85,B 0,C 180,E1 -18538.432,E2 -18538.432} C_VEL
LIN {X 0,Y 256.71,Z 527.483,A -85,B 0,C 180,E1 -18541.569,E2 -18541.569} C_VEL
LIN {X 0,Y 256.467,Z 527.517,A -85,B 0,C 180,E1 -18546.72,E2 -18546.72} C_VEL
LIN {X 0,Y 256.422,Z 527.517,A -85,B 0,C 180,E1 -18549.466,E2 -18549.466} C_VEL
LIN {X 0,Y 256.246,Z 527.553,A -85,B 0,C 180,E1 -18554.291,E2 -18554.291} C_VEL
LIN {X 0,Y 256.199,Z 527.55,A -85,B 0,C 180,E1 -18557.563,E2 -18557.563} C_VEL
LIN {X 0,Y 256.153,Z 527.571,A -85,B 0,C 180,E1 -18561.12,E2 -18561.12} C_VEL
LIN {X 0,Y 256.185,Z 527.563,A -85,B 0,C 180,E1 -18565.14,E2 -18565.14} C_VEL
LIN {X 0,Y 256.113,Z 527.563,A -85,B 0,C 180,E1 -18569.6,E2 -18569.6} C_VEL
LIN {X 0,Y 256.065,Z 527.585,A -85,B 0,C 180,E1 -18573.294,E2 -18573.294} C_VEL
LIN {X 0,Y 256.113,Z 527.588,A -85,B 0,C 180,E1 -18577.272,E2 -18577.272} C_VEL
LIN {X 0,Y 256.054,Z 527.594,A -85,B 0,C 180,E1 -18581.204,E2 -18581.204} C_VEL
LIN {X 0,Y 256.061,Z 527.593,A -85,B 0,C 180,E1 -18585.53,E2 -18585.53} C_VEL
LIN {X 0,Y 256.116,Z 527.676,A -85,B 0,C 180,E1 -18588.61,E2 -18588.61} C_VEL
LIN {X 0,Y 260.223,Z 540.567,A -85,B 0,C 180,E1 -18592.779,E2 -18592.779} C_VEL
LIN {X 0,Y 263.026,Z 551.13,A -85,B 0,C 180,E1 -18595.868,E2 -18595.868} C_VEL
LIN {X 0,Y 270.723,Z 568.177,A -85,B 0,C 180,E1 -18597.448,E2 -18597.448} C_VEL
LIN {X 0,Y 271.807,Z 571.629,A -85,B 0,C 180,E1 -18597.693,E2 -18597.693} C_VEL
LIN {X 0,Y 275.007,Z 589.855,A -85,B 0,C 180,E1 -18598.641,E2 -18598.641} C_VEL
LIN {X 0,Y 272.442,Z 661.967,A -85,B 0,C 180,E1 -18600.514,E2 -18600.514} C_VEL
LIN {X 0,Y 271.457,Z 675.126,A -85,B 0,C 180,E1 -18601.119,E2 -18601.119} C_VEL
LIN {X 0,Y 270.202,Z 687.252,A -85,B 0,C 180,E1 -18601.979,E2 -18601.979} C_VEL
LIN {X 0,Y 268.619,Z 699.151,A -85,B 0,C 180,E1 -18603.124,E2 -18603.124} C_VEL
LIN {X 0,Y 266.783,Z 709.856,A -85,B 0,C 180,E1 -18604.446,E2 -18604.446} C_VEL
LIN {X 0,Y 264.61,Z 720.431,A -85,B 0,C 180,E1 -18606.107,E2 -18606.107} C_VEL
LIN {X 0,Y 262.449,Z 729.944,A -85,B 0,C 180,E1 -18607.983,E2 -18607.983} C_VEL
LIN {X 0,Y 260.534,Z 737.737,A -85,B 0,C 180,E1 -18609.884,E2 -18609.884} C_VEL
LIN {X 0,Y 258.813,Z 745.013,A -85,B 0,C 180,E1 -18612.088,E2 -18612.088} C_VEL
LIN {X 0,Y 257.538,Z 750.529,A -85,B 0,C 180,E1 -18614.164,E2 -18614.164} C_VEL
LIN {X 0,Y 256.134,Z 755.54,A -85,B 0,C 180,E1 -18616.513,E2 -18616.513} C_VEL
LIN {X 0,Y 255.246,Z 759.397,A -85,B 0,C 180,E1 -18618.888,E2 -18618.888} C_VEL
LIN {X 0,Y 254.793,Z 761.371,A -85,B 0,C 180,E1 -18620.474,E2 -18620.474} C_VEL
LIN {X 0,Y 254.438,Z 762.937,A -85,B 0,C 180,E1 -18622.062,E2 -18622.062} C_VEL
LIN {X 0,Y 254.088,Z 764.633,A -85,B 0,C 180,E1 -18624.723,E2 -18624.723} C_VEL
LIN {X 0,Y 254.048,Z 765.152,A -85,B 0,C 180,E1 -18626.828,E2 -18626.828} C_VEL
LIN {X 0,Y 254.041,Z 765.108,A -85,B 0,C 180,E1 -18628.415,E2 -18628.415} C_VEL
LIN {X 0,Y 254.06,Z 764.671,A -85,B 0,C 180,E1 -18630,E2 -18630} C_VEL
LIN {X 0,Y 254.36,Z 762.549,A -85,B 0,C 180,E1 -18633.168,E2 -18633.168} C_VEL
LIN {X 0,Y 254.8,Z 759.881,A -85,B 0,C 180,E1 -18635.54,E2 -18635.54} C_VEL
LIN {X 0,Y 255.38,Z 756.207,A -85,B 0,C 180,E1 -18637.909,E2 -18637.909} C_VEL
LIN {X 0,Y 256.319,Z 751.419,A -85,B 0,C 180,E1 -18640.266,E2 -18640.266} C_VEL
LIN {X 0,Y 257.582,Z 745.376,A -85,B 0,C 180,E1 -18642.607,E2 -18642.607} C_VEL
LIN {X 0,Y 259.21,Z 737.816,A -85,B 0,C 180,E1 -18644.926,E2 -18644.926} C_VEL
LIN {X 0,Y 261.2,Z 728.341,A -85,B 0,C 180,E1 -18647.215,E2 -18647.215} C_VEL
LIN {X 0,Y 263.073,Z 718.546,A -85,B 0,C 180,E1 -18649.102,E2 -18649.102} C_VEL
LIN {X 0,Y 265.018,Z 707.492,A -85,B 0,C 180,E1 -18650.774,E2 -18650.774} C_VEL
LIN {X 0,Y 266.545,Z 696.707,A -85,B 0,C 180,E1 -18652.069,E2 -18652.069} C_VEL
LIN {X 0,Y 267.983,Z 685.89,A -85,B 0,C 180,E1 -18653.062,E2 -18653.062} C_VEL
LIN {X 0,Y 268.956,Z 673.821,A -85,B 0,C 180,E1 -18653.906,E2 -18653.906} C_VEL
LIN {X 0,Y 269.836,Z 659.753,A -85,B 0,C 180,E1 -18654.527,E2 -18654.527} C_VEL
LIN {X 0,Y 272.065,Z 587.476,A -85,B 0,C 180,E1 -18656.415,E2 -18656.415} C_VEL
LIN {X 0,Y 268.249,Z 565.012,A -85,B 0,C 180,E1 -18657.512,E2 -18657.512} C_VEL
LIN {X 0,Y 262.57,Z 550.846,A -85,B 0,C 180,E1 -18658.672,E2 -18658.672} C_VEL
LIN {X 0,Y 259.344,Z 538.453,A -85,B 0,C 180,E1 -18662.152,E2 -18662.152} C_VEL
LIN {X 0,Y 256.134,Z 527.578,A -85,B 0,C 180,E1 -18665.545,E2 -18665.545} C_VEL
LIN {X 0,Y 256.131,Z 527.57,A -85,B 0,C 180,E1 -18669.798,E2 -18669.798} C_VEL
LIN {X 0,Y 256.103,Z 527.582,A -85,B 0,C 180,E1 -18673.317,E2 -18673.317} C_VEL
LIN {X 0,Y 256.108,Z 527.579,A -85,B 0,C 180,E1 -18677.128,E2 -18677.128} C_VEL
LIN {X 0,Y 266.064,Z 556.391,A -85,B 0,C 180,E1 -18678.942,E2 -18678.942} C_VEL
LIN {X 0,Y 263.344,Z 625.016,A -85,B 0,C 180,E1 -18681.465,E2 -18681.465} C_VEL
LIN {X 0,Y 262.666,Z 638.664,A -85,B 0,C 180,E1 -18682.261,E2 -18682.261} C_VEL
LIN {X 0,Y 261.731,Z 651.521,A -85,B 0,C 180,E1 -18683.311,E2 -18683.311} C_VEL
LIN {X 0,Y 260.794,Z 662.011,A -85,B 0,C 180,E1 -18684.424,E2 -18684.424} C_VEL
LIN {X 0,Y 259.7,Z 667.158,A -85,B 0,C 180,E1 -18685.042,E2 -18685.042} C_VEL
LIN {X 0,Y 256.08,Z 675.127,A -85,B 0,C 180,E1 -18686.072,E2 -18686.072} C_VEL
LIN {X 0,Y 252.386,Z 682.736,A -85,B 0,C 180,E1 -18687.243,E2 -18687.243} C_VEL
LIN {X 0,Y 251.19,Z 687.217,A -85,B 0,C 180,E1 -18688.072,E2 -18688.072} C_VEL
LIN {X 0,Y 249.986,Z 697.136,A -85,B 0,C 180,E1 -18690.25,E2 -18690.25} C_VEL
LIN {X 0,Y 248.992,Z 706.019,A -85,B 0,C 180,E1 -18692.698,E2 -18692.698} C_VEL
LIN {X 0,Y 248.285,Z 713.634,A -85,B 0,C 180,E1 -18695.322,E2 -18695.322} C_VEL
LIN {X 0,Y 247.758,Z 718.622,A -85,B 0,C 180,E1 -18697.483,E2 -18697.483} C_VEL
LIN {X 0,Y 247.423,Z 723.325,A -85,B 0,C 180,E1 -18700.07,E2 -18700.07} C_VEL
LIN {X 0,Y 247.28,Z 725.724,A -85,B 0,C 180,E1 -18701.781,E2 -18701.781} C_VEL
LIN {X 0,Y 247.299,Z 727.657,A -85,B 0,C 180,E1 -18703.489,E2 -18703.489} C_VEL
LIN {X 0,Y 247.463,Z 729.089,A -85,B 0,C 180,E1 -18705.19,E2 -18705.19} C_VEL
LIN {X 0,Y 247.699,Z 730.043,A -85,B 0,C 180,E1 -18706.88,E2 -18706.88} C_VEL
LIN {X 0,Y 248.06,Z 730.574,A -85,B 0,C 180,E1 -18708.561,E2 -18708.561} C_VEL
LIN {X 0,Y 248.942,Z 730.488,A -85,B 0,C 180,E1 -18711.144,E2 -18711.144} C_VEL
LIN {X 0,Y 249.997,Z 729.461,A -85,B 0,C 180,E1 -18713.543,E2 -18713.543} C_VEL
LIN {X 0,Y 250.94,Z 728.238,A -85,B 0,C 180,E1 -18715.18,E2 -18715.18} C_VEL
LIN {X 0,Y 253.123,Z 724.625,A -85,B 0,C 180,E1 -18718.23,E2 -18718.23} C_VEL
LIN {X 0,Y 255.4,Z 720.217,A -85,B 0,C 180,E1 -18720.788,E2 -18720.788} C_VEL
LIN {X 0,Y 258.342,Z 713.893,A -85,B 0,C 180,E1 -18723.509,E2 -18723.509} C_VEL
LIN {X 0,Y 261.38,Z 706.772,A -85,B 0,C 180,E1 -18725.826,E2 -18725.826} C_VEL
LIN {X 0,Y 264.644,Z 698.242,A -85,B 0,C 180,E1 -18728.014,E2 -18728.014} C_VEL
LIN {X 0,Y 267.939,Z 688.466,A -85,B 0,C 180,E1 -18730.007,E2 -18730.007} C_VEL
LIN {X 0,Y 271.272,Z 677.404,A -85,B 0,C 180,E1 -18731.772,E2 -18731.772} C_VEL
LIN {X 0,Y 274.405,Z 664.787,A -85,B 0,C 180,E1 -18733.327,E2 -18733.327} C_VEL
LIN {X 0,Y 276.909,Z 652.287,A -85,B 0,C 180,E1 -18734.523,E2 -18734.523} C_VEL
LIN {X 0,Y 278.995,Z 638.733,A -85,B 0,C 180,E1 -18735.49,E2 -18735.49} C_VEL
LIN {X 0,Y 280.42,Z 625.507,A -85,B 0,C 180,E1 -18736.137,E2 -18736.137} C_VEL
LIN {X 0,Y 285.207,Z 579.891,A -85,B 0,C 180,E1 -18737.945,E2 -18737.945} C_VEL
LIN {X 0,Y 281.607,Z 573.083,A -85,B 0,C 180,E1 -18739.54,E2 -18739.54} C_VEL
LIN {X 0,Y 277.986,Z 567.225,A -85,B 0,C 180,E1 -18741.29,E2 -18741.29} C_VEL
LIN {X 0,Y 275.264,Z 563.267,A -85,B 0,C 180,E1 -18742.748,E2 -18742.748} C_VEL
